KUKA KRL program: EPS_2_25694_RR02_A_20251117072404.src

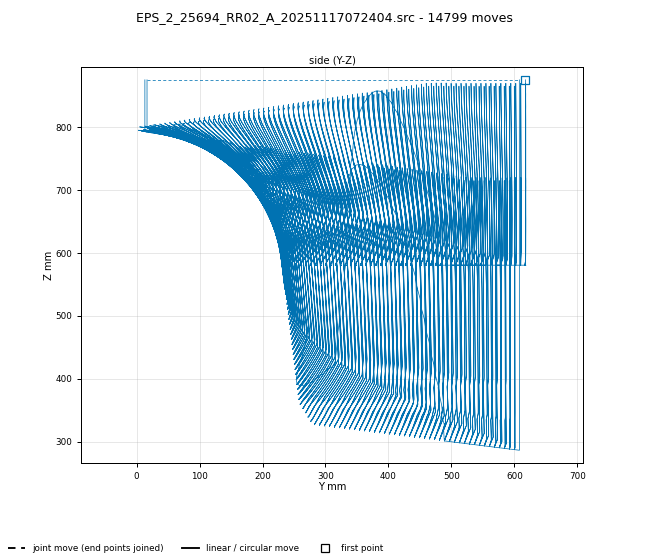
[picture p0: tool path of EPS_2_25694_RR02_A_20251117072404.src, 14799 of 14801 moves have a stored position in this frame; points joined in program order, loops and branches not executed]
&ACCESS RVP
&REL 4
&COMMENT QRS 19112012
&PARAM EDITMASK = *
DEF PART()
EXT BAS (BAS_COMMAND :IN,REAL :IN )
INT I
BAS (#INITMOV,0 )

;KUKA QRS Post kuka4.cps  Date:22-06-2017 !

File_ID=2908

QRS_PRE_INIT()

;Init var - Until changes are made in qrs_pre_init
Outlet_Square_prg=0
Inlet_1_Square_prg=0
Inlet_2_Square_prg=0
Inlet_3_Square_prg=0
Inlet_4_Square_prg=0
Inlet_5_Square_prg=0

Outlet_1={X 0.000, Y 466.000, Z 636.500, B 0.000, E1 0.000 }
Inlet_1={X 0.000, Y 521.440, Z 392.000, B 0.000, E1 180.000 }
Outlet_1_type=457
Inlet_1_type=366
;QRS#1=Sidecore dimensions
;QRS#2=450-18" Concrete
;QRS#3=375-15" PVC SDR 35
;QRS#4=
;QRS#5=
;QRS#6=
;QRS#7=
;QRS#8=
;QRS#9=28A PSX-2
;QRS#10=20Y PSX
;QRS#11=
;QRS#12=
;QRS#13=
;QRS#14=
;QRS#15=
;QRS#16=1220x127x1219 4'
;QRS#17=EPS Height
;QRS#18=865
;QRS#19=*
;QRS#20= UPDATED VERSION 22-06-2017
;QRS#21=*
Outlet_Square=0250
Inlet_1_Square=0250
Inlet_2_Square=0
Inlet_3_Square=0
Inlet_4_Square=0
Inlet_5_Square=0
Mill_Square=1
Outlet_Square_Prg=274
Inlet_1_Square_prg=252

QRS_INIT()

$ADVANCE=5

; T1
PTP {E1 171.23,E2 171.23}
PTP {X 0,Y 617.527,A -85,B 0,C 180,E1 171.23,E2 171.23,E3 0,E4 0,E5 0,E6 0}
QRS_SPEED_INIT()
LIN {X 0,Y 617.527,Z 875,A -85,B 0,C 180,E1 171.23,E2 171.23,E3 0,E4 0,E5 0,E6 0} C_VEL
LIN {X 0,Y 617.527,Z 582.66,A -85,B 0,C 180,E1 171.23,E2 171.23} C_VEL
LIN {X 0,Y 617.508,Z 580.66,A -85,B 0,C 180,E1 171.416,E2 171.416} C_VEL
LIN {X 0,Y 618.008,Z 580.66,A -85,B 0,C 180,E1 174.214,E2 174.214} C_VEL
LIN {X 0,Y 618.036,Z 580.66,A -85,B 0,C 180,E1 178.845,E2 178.845} C_VEL
LIN {X 0,Y 617.997,Z 580.66,A -85,B 0,C 180,E1 183.468,E2 183.468} C_VEL
LIN {X 0,Y 618.006,Z 580.66,A -85,B 0,C 180,E1 188.114,E2 188.114} C_VEL
LIN {X 0,Y 617.984,Z 580.66,A -85,B 0,C 180,E1 192.815,E2 192.815} C_VEL
LIN {X 0,Y 617.935,Z 580.66,A -85,B 0,C 180,E1 197.607,E2 197.607} C_VEL
LIN {X 0,Y 617.752,Z 580.66,A -85,B 0,C 180,E1 198.547,E2 198.547} C_VEL
LIN {X 0,Y 617.939,Z 580.66,A -85,B 0,C 180,E1 202.529,E2 202.529} C_VEL
LIN {X 0,Y 617.436,Z 580.66,A -85,B 0,C 180,E1 205.077,E2 205.077} C_VEL
LIN {X 0,Y 617.874,Z 580.66,A -85,B 0,C 180,E1 207.637,E2 207.637} C_VEL
LIN {X 0,Y 617.365,Z 580.66,A -85,B 0,C 180,E1 210.306,E2 210.306} C_VEL
LIN {X 0,Y 617.833,Z 580.66,A -85,B 0,C 180,E1 212.996,E2 212.996} C_VEL
LIN {X 0,Y 617.707,Z 580.66,A -85,B 0,C 180,E1 214.198,E2 214.198} C_VEL
LIN {X 0,Y 617.789,Z 580.66,A -85,B 0,C 180,E1 218.704,E2 218.704} C_VEL
LIN {X 0,Y 617.444,Z 580.66,A -85,B 0,C 180,E1 221.76,E2 221.76} C_VEL
LIN {X 0,Y 617.867,Z 580.66,A -85,B 0,C 180,E1 224.902,E2 224.902} C_VEL
LIN {X 0,Y 617.783,Z 580.66,A -85,B 0,C 180,E1 228.274,E2 228.274} C_VEL
LIN {X 0,Y 617.565,Z 580.66,A -85,B 0,C 180,E1 231.28,E2 231.28} C_VEL
LIN {X 0,Y 617.589,Z 580.66,A -85,B 0,C 180,E1 231.899,E2 231.899} C_VEL
LIN {X 0,Y 617.827,Z 580.66,A -85,B 0,C 180,E1 234.204,E2 234.204} C_VEL
LIN {X 0,Y 617.354,Z 580.66,A -85,B 0,C 180,E1 236.976,E2 236.976} C_VEL
LIN {X 0,Y 617.913,Z 580.66,A -85,B 0,C 180,E1 239.724,E2 239.724} C_VEL
LIN {X 0,Y 617.932,Z 580.66,A -85,B 0,C 180,E1 243.987,E2 243.987} C_VEL
LIN {X 0,Y 617.833,Z 580.66,A -85,B 0,C 180,E1 244.426,E2 244.426} C_VEL
LIN {X 0,Y 617.179,Z 580.66,A -85,B 0,C 180,E1 244.545,E2 244.545} C_VEL
LIN {X 0,Y 616.44,Z 580.66,A -85,B 0,C 180,E1 244.616,E2 244.616} C_VEL
LIN {X 0,Y 617.56,Z 586.788,A -85,B 0,C 180,E1 244.746,E2 244.746} C_VEL
LIN {X 0,Y 617.714,Z 589.526,A -85,B 0,C 180,E1 244.787,E2 244.787} C_VEL
LIN {X 0,Y 617.934,Z 647.055,A -85,B 0,C 180,E1 245.527,E2 245.527} C_VEL
LIN {X 0,Y 617.874,Z 657.74,A -85,B 0,C 180,E1 245.698,E2 245.698} C_VEL
LIN {X 0,Y 617.784,Z 666.504,A -85,B 0,C 180,E1 245.868,E2 245.868} C_VEL
LIN {X 0,Y 617.891,Z 680.089,A -85,B 0,C 180,E1 246.215,E2 246.215} C_VEL
LIN {X 0,Y 617.826,Z 690.542,A -85,B 0,C 180,E1 246.526,E2 246.526} C_VEL
LIN {X 0,Y 617.931,Z 702.898,A -85,B 0,C 180,E1 246.968,E2 246.968} C_VEL
LIN {X 0,Y 617.943,Z 713.369,A -85,B 0,C 180,E1 247.393,E2 247.393} C_VEL
LIN {X 0,Y 617.876,Z 723.673,A -85,B 0,C 180,E1 247.859,E2 247.859} C_VEL
LIN {X 0,Y 617.946,Z 734.342,A -85,B 0,C 180,E1 248.407,E2 248.407} C_VEL
LIN {X 0,Y 617.967,Z 745.217,A -85,B 0,C 180,E1 249.027,E2 249.027} C_VEL
LIN {X 0,Y 617.938,Z 755.025,A -85,B 0,C 180,E1 249.644,E2 249.644} C_VEL
LIN {X 0,Y 617.951,Z 764.531,A -85,B 0,C 180,E1 250.302,E2 250.302} C_VEL
LIN {X 0,Y 617.956,Z 773.726,A -85,B 0,C 180,E1 250.999,E2 250.999} C_VEL
LIN {X 0,Y 617.961,Z 782.652,A -85,B 0,C 180,E1 251.74,E2 251.74} C_VEL
LIN {X 0,Y 617.941,Z 791.031,A -85,B 0,C 180,E1 252.497,E2 252.497} C_VEL
LIN {X 0,Y 617.896,Z 798.423,A -85,B 0,C 180,E1 253.221,E2 253.221} C_VEL
LIN {X 0,Y 617.951,Z 806.122,A -85,B 0,C 180,E1 254.046,E2 254.046} C_VEL
LIN {X 0,Y 617.974,Z 812.663,A -85,B 0,C 180,E1 254.803,E2 254.803} C_VEL
LIN {X 0,Y 617.884,Z 819.775,A -85,B 0,C 180,E1 255.697,E2 255.697} C_VEL
LIN {X 0,Y 617.866,Z 826.241,A -85,B 0,C 180,E1 256.589,E2 256.589} C_VEL
LIN {X 0,Y 617.965,Z 832.101,A -85,B 0,C 180,E1 257.481,E2 257.481} C_VEL
LIN {X 0,Y 617.876,Z 837.462,A -85,B 0,C 180,E1 258.365,E2 258.365} C_VEL
LIN {X 0,Y 617.831,Z 843.765,A -85,B 0,C 180,E1 259.541,E2 259.541} C_VEL
LIN {X 0,Y 617.913,Z 847.328,A -85,B 0,C 180,E1 260.28,E2 260.28} C_VEL
LIN {X 0,Y 617.929,Z 852.365,A -85,B 0,C 180,E1 261.45,E2 261.45} C_VEL
LIN {X 0,Y 617.83,Z 855.756,A -85,B 0,C 180,E1 262.35,E2 262.35} C_VEL
LIN {X 0,Y 617.936,Z 860.149,A -85,B 0,C 180,E1 263.748,E2 263.748} C_VEL
LIN {X 0,Y 617.913,Z 862.617,A -85,B 0,C 180,E1 264.677,E2 264.677} C_VEL
LIN {X 0,Y 617.79,Z 864.668,A -85,B 0,C 180,E1 265.604,E2 265.604} C_VEL
LIN {X 0,Y 617.81,Z 866.258,A -85,B 0,C 180,E1 266.531,E2 266.531} C_VEL
LIN {X 0,Y 617.946,Z 867.44,A -85,B 0,C 180,E1 267.457,E2 267.457} C_VEL
LIN {X 0,Y 617.798,Z 868.661,A -85,B 0,C 180,E1 268.844,E2 268.844} C_VEL
LIN {X 0,Y 617.834,Z 868.908,A -85,B 0,C 180,E1 270.231,E2 270.231} C_VEL
LIN {X 0,Y 617.983,Z 868.61,A -85,B 0,C 180,E1 271.155,E2 271.155} C_VEL
LIN {X 0,Y 617.848,Z 867.993,A -85,B 0,C 180,E1 272.08,E2 272.08} C_VEL
LIN {X 0,Y 617.842,Z 866.25,A -85,B 0,C 180,E1 273.469,E2 273.469} C_VEL
LIN {X 0,Y 617.982,Z 864.618,A -85,B 0,C 180,E1 274.394,E2 274.394} C_VEL
LIN {X 0,Y 617.84,Z 862.637,A -85,B 0,C 180,E1 275.323,E2 275.323} C_VEL
LIN {X 0,Y 617.779,Z 860.19,A -85,B 0,C 180,E1 276.253,E2 276.253} C_VEL
LIN {X 0,Y 617.946,Z 855.729,A -85,B 0,C 180,E1 277.648,E2 277.648} C_VEL
LIN {X 0,Y 617.875,Z 851.344,A -85,B 0,C 180,E1 278.796,E2 278.796} C_VEL
LIN {X 0,Y 617.822,Z 847.617,A -85,B 0,C 180,E1 279.666,E2 279.666} C_VEL
LIN {X 0,Y 617.935,Z 842.259,A -85,B 0,C 180,E1 280.75,E2 280.75} C_VEL
LIN {X 0,Y 617.942,Z 837.451,A -85,B 0,C 180,E1 281.633,E2 281.633} C_VEL
LIN {X 0,Y 617.865,Z 830.2,A -85,B 0,C 180,E1 282.817,E2 282.817} C_VEL
LIN {X 0,Y 617.941,Z 824.139,A -85,B 0,C 180,E1 283.706,E2 283.706} C_VEL
LIN {X 0,Y 617.959,Z 817.472,A -85,B 0,C 180,E1 284.599,E2 284.599} C_VEL
LIN {X 0,Y 617.884,Z 809.504,A -85,B 0,C 180,E1 285.571,E2 285.571} C_VEL
LIN {X 0,Y 617.919,Z 802.445,A -85,B 0,C 180,E1 286.357,E2 286.357} C_VEL
LIN {X 0,Y 617.971,Z 794.292,A -85,B 0,C 180,E1 287.188,E2 287.188} C_VEL
LIN {X 0,Y 617.933,Z 787.152,A -85,B 0,C 180,E1 287.863,E2 287.863} C_VEL
LIN {X 0,Y 617.924,Z 778.254,A -85,B 0,C 180,E1 288.634,E2 288.634} C_VEL
LIN {X 0,Y 617.944,Z 769.358,A -85,B 0,C 180,E1 289.339,E2 289.339} C_VEL
LIN {X 0,Y 617.96,Z 760.867,A -85,B 0,C 180,E1 289.959,E2 289.959} C_VEL
LIN {X 0,Y 617.948,Z 751.476,A -85,B 0,C 180,E1 290.587,E2 290.587} C_VEL
LIN {X 0,Y 617.918,Z 741.285,A -85,B 0,C 180,E1 291.206,E2 291.206} C_VEL
LIN {X 0,Y 617.943,Z 731.422,A -85,B 0,C 180,E1 291.749,E2 291.749} C_VEL
LIN {X 0,Y 617.958,Z 720.367,A -85,B 0,C 180,E1 292.293,E2 292.293} C_VEL
LIN {X 0,Y 617.922,Z 709.607,A -85,B 0,C 180,E1 292.767,E2 292.767} C_VEL
LIN {X 0,Y 617.801,Z 699.701,A -85,B 0,C 180,E1 293.16,E2 293.16} C_VEL
LIN {X 0,Y 617.928,Z 686.719,A -85,B 0,C 180,E1 293.589,E2 293.589} C_VEL
LIN {X 0,Y 617.909,Z 674.953,A -85,B 0,C 180,E1 293.921,E2 293.921} C_VEL
LIN {X 0,Y 617.766,Z 663.559,A -85,B 0,C 180,E1 294.193,E2 294.193} C_VEL
LIN {X 0,Y 617.92,Z 651.868,A -85,B 0,C 180,E1 294.402,E2 294.402} C_VEL
LIN {X 0,Y 617.892,Z 634.191,A -85,B 0,C 180,E1 294.645,E2 294.645} C_VEL
LIN {X 0,Y 617.601,Z 587.358,A -85,B 0,C 180,E1 295.246,E2 295.246} C_VEL
LIN {X 0,Y 616.593,Z 581.43,A -85,B 0,C 180,E1 295.365,E2 295.365} C_VEL
LIN {X 0,Y 616.475,Z 580.66,A -85,B 0,C 180,E1 295.385,E2 295.385} C_VEL
LIN {X 0,Y 617.979,Z 580.66,A -85,B 0,C 180,E1 295.627,E2 295.627} C_VEL
LIN {X 0,Y 617.998,Z 580.66,A -85,B 0,C 180,E1 297.63,E2 297.63} C_VEL
LIN {X 0,Y 617.388,Z 580.66,A -85,B 0,C 180,E1 300.304,E2 300.304} C_VEL
LIN {X 0,Y 617.846,Z 580.66,A -85,B 0,C 180,E1 302.994,E2 302.994} C_VEL
LIN {X 0,Y 617.706,Z 580.66,A -85,B 0,C 180,E1 304.196,E2 304.196} C_VEL
LIN {X 0,Y 617.791,Z 580.66,A -85,B 0,C 180,E1 308.702,E2 308.702} C_VEL
LIN {X 0,Y 617.444,Z 580.66,A -85,B 0,C 180,E1 311.758,E2 311.758} C_VEL
LIN {X 0,Y 617.868,Z 580.66,A -85,B 0,C 180,E1 314.9,E2 314.9} C_VEL
LIN {X 0,Y 617.801,Z 580.66,A -85,B 0,C 180,E1 318.269,E2 318.269} C_VEL
LIN {X 0,Y 617.562,Z 580.66,A -85,B 0,C 180,E1 321.279,E2 321.279} C_VEL
LIN {X 0,Y 617.588,Z 580.66,A -85,B 0,C 180,E1 321.896,E2 321.896} C_VEL
LIN {X 0,Y 617.813,Z 580.66,A -85,B 0,C 180,E1 324.202,E2 324.202} C_VEL
LIN {X 0,Y 617.354,Z 580.66,A -85,B 0,C 180,E1 326.975,E2 326.975} C_VEL
LIN {X 0,Y 617.895,Z 580.66,A -85,B 0,C 180,E1 329.723,E2 329.723} C_VEL
LIN {X 0,Y 617.412,Z 580.66,A -85,B 0,C 180,E1 332.341,E2 332.341} C_VEL
LIN {X 0,Y 617.889,Z 580.66,A -85,B 0,C 180,E1 334.943,E2 334.943} C_VEL
LIN {X 0,Y 617.435,Z 580.66,A -85,B 0,C 180,E1 337.451,E2 337.451} C_VEL
LIN {X 0,Y 617.94,Z 580.66,A -85,B 0,C 180,E1 339.951,E2 339.951} C_VEL
LIN {X 0,Y 618.042,Z 580.66,A -85,B 0,C 180,E1 343.627,E2 343.627} C_VEL
LIN {X 0,Y 617.994,Z 580.66,A -85,B 0,C 180,E1 349.544,E2 349.544} C_VEL
LIN {X 0,Y 617.978,Z 580.66,A -85,B 0,C 180,E1 354.213,E2 354.213} C_VEL
LIN {X 0,Y 618.008,Z 580.66,A -85,B 0,C 180,E1 358.845,E2 358.845} C_VEL
LIN {X 0,Y 618.048,Z 580.66,A -85,B 0,C 180,E1 363.468,E2 363.468} C_VEL
LIN {X 0,Y 617.988,Z 580.66,A -85,B 0,C 180,E1 368.114,E2 368.114} C_VEL
LIN {X 0,Y 617.946,Z 580.66,A -85,B 0,C 180,E1 372.816,E2 372.816} C_VEL
LIN {X 0,Y 617.967,Z 580.66,A -85,B 0,C 180,E1 377.606,E2 377.606} C_VEL
LIN {X 0,Y 617.768,Z 580.66,A -85,B 0,C 180,E1 378.552,E2 378.552} C_VEL
LIN {X 0,Y 617.894,Z 580.66,A -85,B 0,C 180,E1 382.531,E2 382.531} C_VEL
LIN {X 0,Y 617.414,Z 580.66,A -85,B 0,C 180,E1 385.078,E2 385.078} C_VEL
LIN {X 0,Y 617.881,Z 580.66,A -85,B 0,C 180,E1 387.637,E2 387.637} C_VEL
LIN {X 0,Y 617.423,Z 580.66,A -85,B 0,C 180,E1 390.303,E2 390.303} C_VEL
LIN {X 0,Y 617.948,Z 580.66,A -85,B 0,C 180,E1 392.989,E2 392.989} C_VEL
LIN {X 0,Y 617.682,Z 580.66,A -85,B 0,C 180,E1 395.807,E2 395.807} C_VEL
LIN {X 0,Y 617.691,Z 580.66,A -85,B 0,C 180,E1 398.116,E2 398.116} C_VEL
LIN {X 0,Y 617.801,Z 580.66,A -85,B 0,C 180,E1 401.731,E2 401.731} C_VEL
LIN {X 0,Y 617.417,Z 580.66,A -85,B 0,C 180,E1 405.059,E2 405.059} C_VEL
LIN {X 0,Y 617.803,Z 580.66,A -85,B 0,C 180,E1 408.271,E2 408.271} C_VEL
LIN {X 0,Y 617.697,Z 580.66,A -85,B 0,C 180,E1 411.886,E2 411.886} C_VEL
LIN {X 0,Y 617.736,Z 580.66,A -85,B 0,C 180,E1 414.198,E2 414.198} C_VEL
LIN {X 0,Y 617.843,Z 580.66,A -85,B 0,C 180,E1 415.785,E2 415.785} C_VEL
LIN {X 0,Y 617.877,Z 580.66,A -85,B 0,C 180,E1 417.008,E2 417.008} C_VEL
LIN {X 0,Y 617.647,Z 580.66,A -85,B 0,C 180,E1 420.175,E2 420.175} C_VEL
LIN {X 0,Y 617.665,Z 580.66,A -85,B 0,C 180,E1 422.354,E2 422.354} C_VEL
LIN {X 0,Y 617.522,Z 580.66,A -85,B 0,C 180,E1 425.242,E2 425.242} C_VEL
LIN {X 0,Y 617.828,Z 580.66,A -85,B 0,C 180,E1 427.467,E2 427.467} C_VEL
LIN {X 0,Y 618.012,Z 580.66,A -85,B 0,C 180,E1 430.997,E2 430.997} C_VEL
LIN {X 0,Y 617.801,Z 580.749,A -85,B 0,C 180,E1 431.084,E2 431.084} C_VEL
LIN {X 0,Y 617.923,Z 591.91,A -85,B 0,C 180,E1 431.53,E2 431.53} C_VEL
LIN {X 0,Y 617.91,Z 600.741,A -85,B 0,C 180,E1 431.928,E2 431.928} C_VEL
LIN {X 0,Y 617.976,Z 609.876,A -85,B 0,C 180,E1 432.395,E2 432.395} C_VEL
LIN {X 0,Y 617.992,Z 617.77,A -85,B 0,C 180,E1 432.84,E2 432.84} C_VEL
LIN {X 0,Y 617.993,Z 624.968,A -85,B 0,C 180,E1 433.284,E2 433.284} C_VEL
LIN {X 0,Y 617.971,Z 633.892,A -85,B 0,C 180,E1 433.895,E2 433.895} C_VEL
LIN {X 0,Y 617.958,Z 641.958,A -85,B 0,C 180,E1 434.505,E2 434.505} C_VEL
LIN {X 0,Y 617.969,Z 649.146,A -85,B 0,C 180,E1 435.102,E2 435.102} C_VEL
LIN {X 0,Y 617.991,Z 655.741,A -85,B 0,C 180,E1 435.7,E2 435.7} C_VEL
LIN {X 0,Y 617.962,Z 663.24,A -85,B 0,C 180,E1 436.443,E2 436.443} C_VEL
LIN {X 0,Y 617.945,Z 670.024,A -85,B 0,C 180,E1 437.184,E2 437.184} C_VEL
LIN {X 0,Y 617.993,Z 677.361,A -85,B 0,C 180,E1 438.072,E2 438.072} C_VEL
LIN {X 0,Y 617.92,Z 683.858,A -85,B 0,C 180,E1 438.955,E2 438.955} C_VEL
LIN {X 0,Y 617.867,Z 688.987,A -85,B 0,C 180,E1 439.728,E2 439.728} C_VEL
LIN {X 0,Y 617.937,Z 694.438,A -85,B 0,C 180,E1 440.656,E2 440.656} C_VEL
LIN {X 0,Y 617.963,Z 698.446,A -85,B 0,C 180,E1 441.413,E2 441.413} C_VEL
LIN {X 0,Y 617.874,Z 702.863,A -85,B 0,C 180,E1 442.351,E2 442.351} C_VEL
LIN {X 0,Y 617.875,Z 704.864,A -85,B 0,C 180,E1 442.817,E2 442.817} C_VEL
LIN {X 0,Y 617.966,Z 708.364,A -85,B 0,C 180,E1 443.749,E2 443.749} C_VEL
LIN {X 0,Y 617.939,Z 711.343,A -85,B 0,C 180,E1 444.678,E2 444.678} C_VEL
LIN {X 0,Y 617.838,Z 713.822,A -85,B 0,C 180,E1 445.605,E2 445.605} C_VEL
LIN {X 0,Y 617.893,Z 715.764,A -85,B 0,C 180,E1 446.532,E2 446.532} C_VEL
LIN {X 0,Y 617.99,Z 717.213,A -85,B 0,C 180,E1 447.458,E2 447.458} C_VEL
LIN {X 0,Y 617.926,Z 717.776,A -85,B 0,C 180,E1 447.92,E2 447.92} C_VEL
LIN {X 0,Y 617.842,Z 718.587,A -85,B 0,C 180,E1 448.845,E2 448.845} C_VEL
LIN {X 0,Y 617.881,Z 718.907,A -85,B 0,C 180,E1 449.769,E2 449.769} C_VEL
LIN {X 0,Y 617.947,Z 718.867,A -85,B 0,C 180,E1 450.231,E2 450.231} C_VEL
LIN {X 0,Y 617.915,Z 718.503,A -85,B 0,C 180,E1 451.156,E2 451.156} C_VEL
LIN {X 0,Y 617.846,Z 717.146,A -85,B 0,C 180,E1 452.543,E2 452.543} C_VEL
LIN {X 0,Y 617.964,Z 715.592,A -85,B 0,C 180,E1 453.468,E2 453.468} C_VEL
LIN {X 0,Y 617.912,Z 713.595,A -85,B 0,C 180,E1 454.395,E2 454.395} C_VEL
LIN {X 0,Y 617.842,Z 711.097,A -85,B 0,C 180,E1 455.323,E2 455.323} C_VEL
LIN {X 0,Y 617.887,Z 708.049,A -85,B 0,C 180,E1 456.252,E2 456.252} C_VEL
LIN {X 0,Y 617.976,Z 704.45,A -85,B 0,C 180,E1 457.182,E2 457.182} C_VEL
LIN {X 0,Y 617.895,Z 700.32,A -85,B 0,C 180,E1 458.116,E2 458.116} C_VEL
LIN {X 0,Y 617.903,Z 695.375,A -85,B 0,C 180,E1 459.084,E2 459.084} C_VEL
LIN {X 0,Y 617.977,Z 690.86,A -85,B 0,C 180,E1 459.867,E2 459.867} C_VEL
LIN {X 0,Y 617.955,Z 687.19,A -85,B 0,C 180,E1 460.456,E2 460.456} C_VEL
LIN {X 0,Y 617.913,Z 682.18,A -85,B 0,C 180,E1 461.192,E2 461.192} C_VEL
LIN {X 0,Y 617.944,Z 676.638,A -85,B 0,C 180,E1 461.929,E2 461.929} C_VEL
LIN {X 0,Y 617.985,Z 670.528,A -85,B 0,C 180,E1 462.667,E2 462.667} C_VEL
LIN {X 0,Y 617.956,Z 663.803,A -85,B 0,C 180,E1 463.409,E2 463.409} C_VEL
LIN {X 0,Y 617.949,Z 657.931,A -85,B 0,C 180,E1 464.004,E2 464.004} C_VEL
LIN {X 0,Y 617.968,Z 651.535,A -85,B 0,C 180,E1 464.599,E2 464.599} C_VEL
LIN {X 0,Y 617.999,Z 644.545,A -85,B 0,C 180,E1 465.196,E2 465.196} C_VEL
LIN {X 0,Y 617.987,Z 637.134,A -85,B 0,C 180,E1 465.777,E2 465.777} C_VEL
LIN {X 0,Y 617.99,Z 628.688,A -85,B 0,C 180,E1 466.378,E2 466.378} C_VEL
LIN {X 0,Y 617.975,Z 620.778,A -85,B 0,C 180,E1 466.888,E2 466.888} C_VEL
LIN {X 0,Y 617.986,Z 613.859,A -85,B 0,C 180,E1 467.298,E2 467.298} C_VEL
LIN {X 0,Y 617.971,Z 605.435,A -85,B 0,C 180,E1 467.75,E2 467.75} C_VEL
LIN {X 0,Y 617.907,Z 596.414,A -85,B 0,C 180,E1 468.184,E2 468.184} C_VEL
LIN {X 0,Y 617.715,Z 586.549,A -85,B 0,C 180,E1 468.606,E2 468.606} C_VEL
LIN {X 0,Y 617.482,Z 580.66,A -85,B 0,C 180,E1 468.848,E2 468.848} C_VEL
LIN {X 0,Y 617.844,Z 580.66,A -85,B 0,C 180,E1 468.93,E2 468.93} C_VEL
LIN {X 0,Y 618.044,Z 580.66,A -85,B 0,C 180,E1 469.031,E2 469.031} C_VEL
LIN {X 0,Y 618.046,Z 580.66,A -85,B 0,C 180,E1 470.045,E2 470.045} C_VEL
LIN {X 0,Y 617.926,Z 580.66,A -85,B 0,C 180,E1 475.055,E2 475.055} C_VEL
LIN {X 0,Y 617.412,Z 580.66,A -85,B 0,C 180,E1 477.659,E2 477.659} C_VEL
LIN {X 0,Y 617.854,Z 580.66,A -85,B 0,C 180,E1 480.279,E2 480.279} C_VEL
LIN {X 0,Y 617.333,Z 580.66,A -85,B 0,C 180,E1 483.025,E2 483.025} C_VEL
LIN {X 0,Y 617.818,Z 580.66,A -85,B 0,C 180,E1 485.797,E2 485.797} C_VEL
LIN {X 0,Y 617.907,Z 580.66,A -85,B 0,C 180,E1 488.694,E2 488.694} C_VEL
LIN {X 0,Y 617.42,Z 580.66,A -85,B 0,C 180,E1 491.761,E2 491.761} C_VEL
LIN {X 0,Y 617.838,Z 580.66,A -85,B 0,C 180,E1 494.903,E2 494.903} C_VEL
LIN {X 0,Y 617.754,Z 580.66,A -85,B 0,C 180,E1 498.275,E2 498.275} C_VEL
LIN {X 0,Y 617.542,Z 580.66,A -85,B 0,C 180,E1 501.278,E2 501.278} C_VEL
LIN {X 0,Y 617.816,Z 580.66,A -85,B 0,C 180,E1 504.202,E2 504.202} C_VEL
LIN {X 0,Y 617.317,Z 580.66,A -85,B 0,C 180,E1 506.973,E2 506.973} C_VEL
LIN {X 0,Y 617.842,Z 580.66,A -85,B 0,C 180,E1 509.72,E2 509.72} C_VEL
LIN {X 0,Y 617.389,Z 580.66,A -85,B 0,C 180,E1 512.339,E2 512.339} C_VEL
LIN {X 0,Y 617.892,Z 580.66,A -85,B 0,C 180,E1 514.943,E2 514.943} C_VEL
LIN {X 0,Y 617.441,Z 580.66,A -85,B 0,C 180,E1 517.452,E2 517.452} C_VEL
LIN {X 0,Y 617.945,Z 580.66,A -85,B 0,C 180,E1 519.951,E2 519.951} C_VEL
LIN {X 0,Y 618.009,Z 580.66,A -85,B 0,C 180,E1 523.636,E2 523.636} C_VEL
LIN {X 0,Y 617.95,Z 580.66,A -85,B 0,C 180,E1 529.543,E2 529.543} C_VEL
LIN {X 0,Y 617.508,Z 580.66,A -85,B 0,C 180,E1 531.416,E2 531.416} C_VEL
LIN {X 0,Y 613.842,Z 580.66,A -85,B 0,C 180,E1 533.008,E2 533.008} C_VEL
LIN {X 0,Y 609.952,Z 580.66,A -85,B 0,C 180,E1 534.619,E2 534.619} C_VEL
LIN {X 0,Y 609.775,Z 580.66,A -85,B 0,C 180,E1 539.996,E2 539.996} C_VEL
LIN {X 0,Y 609.835,Z 580.66,A -85,B 0,C 180,E1 544.267,E2 544.267} C_VEL
LIN {X 0,Y 609.932,Z 580.66,A -85,B 0,C 180,E1 548.561,E2 548.561} C_VEL
LIN {X 0,Y 610.054,Z 580.66,A -85,B 0,C 180,E1 552.902,E2 552.902} C_VEL
LIN {X 0,Y 609.793,Z 580.66,A -85,B 0,C 180,E1 558.826,E2 558.826} C_VEL
LIN {X 0,Y 609.731,Z 580.66,A -85,B 0,C 180,E1 563.405,E2 563.405} C_VEL
LIN {X 0,Y 609.791,Z 580.66,A -85,B 0,C 180,E1 568.143,E2 568.143} C_VEL
LIN {X 0,Y 609.938,Z 580.66,A -85,B 0,C 180,E1 573.095,E2 573.095} C_VEL
LIN {X 0,Y 609.609,Z 580.66,A -85,B 0,C 180,E1 579.652,E2 579.652} C_VEL
LIN {X 0,Y 609.721,Z 580.66,A -85,B 0,C 180,E1 585.949,E2 585.949} C_VEL
LIN {X 0,Y 609.565,Z 580.66,A -85,B 0,C 180,E1 590.345,E2 590.345} C_VEL
LIN {X 0,Y 609.614,Z 580.66,A -85,B 0,C 180,E1 595.163,E2 595.163} C_VEL
LIN {X 0,Y 609.814,Z 580.66,A -85,B 0,C 180,E1 600.331,E2 600.331} C_VEL
LIN {X 0,Y 609.422,Z 580.66,A -85,B 0,C 180,E1 604.278,E2 604.278} C_VEL
LIN {X 0,Y 610.603,Z 601.613,A -85,B 0,C 180,E1 604.626,E2 604.626} C_VEL
LIN {X 0,Y 610.594,Z 666.131,A -85,B 0,C 180,E1 605.557,E2 605.557} C_VEL
LIN {X 0,Y 610.606,Z 702.84,A -85,B 0,C 180,E1 606.673,E2 606.673} C_VEL
LIN {X 0,Y 610.469,Z 736.562,A -85,B 0,C 180,E1 608.254,E2 608.254} C_VEL
LIN {X 0,Y 610.341,Z 768.501,A -85,B 0,C 180,E1 610.345,E2 610.345} C_VEL
LIN {X 0,Y 610.22,Z 797.222,A -85,B 0,C 180,E1 612.863,E2 612.863} C_VEL
LIN {X 0,Y 610.116,Z 822.296,A -85,B 0,C 180,E1 615.814,E2 615.814} C_VEL
LIN {X 0,Y 610.041,Z 841.765,A -85,B 0,C 180,E1 618.909,E2 618.909} C_VEL
LIN {X 0,Y 610.029,Z 856.171,A -85,B 0,C 180,E1 622.153,E2 622.153} C_VEL
LIN {X 0,Y 610.029,Z 864.449,A -85,B 0,C 180,E1 625.015,E2 625.015} C_VEL
LIN {X 0,Y 609.996,Z 869.506,A -85,B 0,C 180,E1 628.576,E2 628.576} C_VEL
LIN {X 0,Y 610.121,Z 869.508,A -85,B 0,C 180,E1 631.421,E2 631.421} C_VEL
LIN {X 0,Y 610.052,Z 864.454,A -85,B 0,C 180,E1 634.982,E2 634.982} C_VEL
LIN {X 0,Y 610.08,Z 853.503,A -85,B 0,C 180,E1 638.562,E2 638.562} C_VEL
LIN {X 0,Y 610.103,Z 836.72,A -85,B 0,C 180,E1 641.994,E2 641.994} C_VEL
LIN {X 0,Y 610.174,Z 815.251,A -85,B 0,C 180,E1 645.103,E2 645.103} C_VEL
LIN {X 0,Y 610.254,Z 788.597,A -85,B 0,C 180,E1 647.972,E2 647.972} C_VEL
LIN {X 0,Y 610.393,Z 758.021,A -85,B 0,C 180,E1 650.413,E2 650.413} C_VEL
LIN {X 0,Y 610.532,Z 725.757,A -85,B 0,C 180,E1 652.315,E2 652.315} C_VEL
LIN {X 0,Y 610.645,Z 690.377,A -85,B 0,C 180,E1 653.772,E2 653.772} C_VEL
LIN {X 0,Y 610.725,Z 653.833,A -85,B 0,C 180,E1 654.679,E2 654.679} C_VEL
LIN {X 0,Y 609.77,Z 584.389,A -85,B 0,C 180,E1 655.631,E2 655.631} C_VEL
LIN {X 0,Y 609.682,Z 580.66,A -85,B 0,C 180,E1 655.757,E2 655.757} C_VEL
LIN {X 0,Y 609.507,Z 580.66,A -85,B 0,C 180,E1 659.787,E2 659.787} C_VEL
LIN {X 0,Y 609.945,Z 580.66,A -85,B 0,C 180,E1 663.097,E2 663.097} C_VEL
LIN {X 0,Y 609.593,Z 580.66,A -85,B 0,C 180,E1 669.658,E2 669.658} C_VEL
LIN {X 0,Y 609.734,Z 580.66,A -85,B 0,C 180,E1 675.957,E2 675.957} C_VEL
LIN {X 0,Y 609.567,Z 580.66,A -85,B 0,C 180,E1 680.349,E2 680.349} C_VEL
LIN {X 0,Y 609.607,Z 580.66,A -85,B 0,C 180,E1 685.169,E2 685.169} C_VEL
LIN {X 0,Y 609.783,Z 580.66,A -85,B 0,C 180,E1 690.341,E2 690.341} C_VEL
LIN {X 0,Y 609.961,Z 580.66,A -85,B 0,C 180,E1 695.045,E2 695.045} C_VEL
LIN {X 0,Y 609.793,Z 580.66,A -85,B 0,C 180,E1 701.174,E2 701.174} C_VEL
LIN {X 0,Y 609.393,Z 580.66,A -85,B 0,C 180,E1 705.678,E2 705.678} C_VEL
LIN {X 0,Y 609.919,Z 580.66,A -85,B 0,C 180,E1 709.997,E2 709.997} C_VEL
LIN {X 0,Y 610.056,Z 580.66,A -85,B 0,C 180,E1 714.307,E2 714.307} C_VEL
LIN {X 0,Y 609.744,Z 580.66,A -85,B 0,C 180,E1 720.004,E2 720.004} C_VEL
LIN {X 0,Y 609.85,Z 580.66,A -85,B 0,C 180,E1 724.275,E2 724.275} C_VEL
LIN {X 0,Y 609.914,Z 580.66,A -85,B 0,C 180,E1 728.57,E2 728.57} C_VEL
LIN {X 0,Y 609.999,Z 580.66,A -85,B 0,C 180,E1 732.912,E2 732.912} C_VEL
LIN {X 0,Y 609.783,Z 580.66,A -85,B 0,C 180,E1 738.835,E2 738.835} C_VEL
LIN {X 0,Y 609.7,Z 580.66,A -85,B 0,C 180,E1 743.415,E2 743.415} C_VEL
LIN {X 0,Y 609.795,Z 580.66,A -85,B 0,C 180,E1 748.152,E2 748.152} C_VEL
LIN {X 0,Y 610.006,Z 580.66,A -85,B 0,C 180,E1 753.1,E2 753.1} C_VEL
LIN {X 0,Y 609.73,Z 580.66,A -85,B 0,C 180,E1 758.378,E2 758.378} C_VEL
LIN {X 0,Y 609.77,Z 580.66,A -85,B 0,C 180,E1 762.103,E2 762.103} C_VEL
LIN {X 0,Y 609.865,Z 580.66,A -85,B 0,C 180,E1 768.145,E2 768.145} C_VEL
LIN {X 0,Y 609.733,Z 580.66,A -85,B 0,C 180,E1 773.422,E2 773.422} C_VEL
LIN {X 0,Y 609.795,Z 580.66,A -85,B 0,C 180,E1 777.59,E2 777.59} C_VEL
LIN {X 0,Y 609.7,Z 580.66,A -85,B 0,C 180,E1 781.85,E2 781.85} C_VEL
LIN {X 0,Y 609.813,Z 580.66,A -85,B 0,C 180,E1 788.137,E2 788.137} C_VEL
LIN {X 0,Y 610.063,Z 580.755,A -85,B 0,C 180,E1 790.836,E2 790.836} C_VEL
LIN {X 0,Y 610.376,Z 612.485,A -85,B 0,C 180,E1 792.312,E2 792.312} C_VEL
LIN {X 0,Y 610.257,Z 642.503,A -85,B 0,C 180,E1 794.338,E2 794.338} C_VEL
LIN {X 0,Y 610.2,Z 667.86,A -85,B 0,C 180,E1 796.733,E2 796.733} C_VEL
LIN {X 0,Y 610.105,Z 688.675,A -85,B 0,C 180,E1 799.456,E2 799.456} C_VEL
LIN {X 0,Y 610.08,Z 704.253,A -85,B 0,C 180,E1 802.397,E2 802.397} C_VEL
LIN {X 0,Y 610.06,Z 713.378,A -85,B 0,C 180,E1 805.018,E2 805.018} C_VEL
LIN {X 0,Y 610.125,Z 717.884,A -85,B 0,C 180,E1 807.157,E2 807.157} C_VEL
LIN {X 0,Y 610.088,Z 719.996,A -85,B 0,C 180,E1 810.001,E2 810.001} C_VEL
LIN {X 0,Y 610.04,Z 717.729,A -85,B 0,C 180,E1 812.846,E2 812.846} C_VEL
LIN {X 0,Y 610.068,Z 709.867,A -85,B 0,C 180,E1 816.056,E2 816.056} C_VEL
LIN {X 0,Y 610.101,Z 697.553,A -85,B 0,C 180,E1 818.924,E2 818.924} C_VEL
LIN {X 0,Y 610.144,Z 679.155,A -85,B 0,C 180,E1 821.814,E2 821.814} C_VEL
LIN {X 0,Y 610.218,Z 655.502,A -85,B 0,C 180,E1 824.441,E2 824.441} C_VEL
LIN {X 0,Y 610.329,Z 627.575,A -85,B 0,C 180,E1 826.669,E2 826.669} C_VEL
LIN {X 0,Y 610.345,Z 595.936,A -85,B 0,C 180,E1 828.439,E2 828.439} C_VEL
LIN {X 0,Y 610.16,Z 580.66,A -85,B 0,C 180,E1 829.133,E2 829.133} C_VEL
LIN {X 0,Y 609.998,Z 580.66,A -85,B 0,C 180,E1 834.959,E2 834.959} C_VEL
LIN {X 0,Y 609.796,Z 580.66,A -85,B 0,C 180,E1 839.775,E2 839.775} C_VEL
LIN {X 0,Y 609.79,Z 580.66,A -85,B 0,C 180,E1 846.577,E2 846.577} C_VEL
LIN {X 0,Y 609.542,Z 580.66,A -85,B 0,C 180,E1 850.228,E2 850.228} C_VEL
LIN {X 0,Y 609.675,Z 580.66,A -85,B 0,C 180,E1 856.07,E2 856.07} C_VEL
LIN {X 0,Y 609.528,Z 580.66,A -85,B 0,C 180,E1 860.357,E2 860.357} C_VEL
LIN {X 0,Y 609.596,Z 580.66,A -85,B 0,C 180,E1 865.158,E2 865.158} C_VEL
LIN {X 0,Y 609.742,Z 580.66,A -85,B 0,C 180,E1 870.353,E2 870.353} C_VEL
LIN {X 0,Y 609.98,Z 580.66,A -85,B 0,C 180,E1 875.038,E2 875.038} C_VEL
LIN {X 0,Y 609.814,Z 580.66,A -85,B 0,C 180,E1 881.166,E2 881.166} C_VEL
LIN {X 0,Y 609.34,Z 580.66,A -85,B 0,C 180,E1 885.708,E2 885.708} C_VEL
LIN {X 0,Y 609.891,Z 580.66,A -85,B 0,C 180,E1 889.989,E2 889.989} C_VEL
LIN {X 0,Y 609.952,Z 580.66,A -85,B 0,C 180,E1 894.619,E2 894.619} C_VEL
LIN {X 0,Y 605.699,Z 580.66,A -85,B 0,C 180,E1 896.215,E2 896.215} C_VEL
LIN {X 0,Y 601.911,Z 580.66,A -85,B 0,C 180,E1 897.833,E2 897.833} C_VEL
LIN {X 0,Y 601.976,Z 580.66,A -85,B 0,C 180,E1 902.879,E2 902.879} C_VEL
LIN {X 0,Y 601.99,Z 580.66,A -85,B 0,C 180,E1 908.675,E2 908.675} C_VEL
LIN {X 0,Y 602.076,Z 580.66,A -85,B 0,C 180,E1 913.076,E2 913.076} C_VEL
LIN {X 0,Y 601.84,Z 580.66,A -85,B 0,C 180,E1 919.085,E2 919.085} C_VEL
LIN {X 0,Y 601.755,Z 580.66,A -85,B 0,C 180,E1 923.734,E2 923.734} C_VEL
LIN {X 0,Y 601.771,Z 580.66,A -85,B 0,C 180,E1 928.552,E2 928.552} C_VEL
LIN {X 0,Y 601.82,Z 580.66,A -85,B 0,C 180,E1 933.879,E2 933.879} C_VEL
LIN {X 0,Y 601.76,Z 580.66,A -85,B 0,C 180,E1 938.971,E2 938.971} C_VEL
LIN {X 0,Y 601.731,Z 580.66,A -85,B 0,C 180,E1 945.208,E2 945.208} C_VEL
LIN {X 0,Y 601.737,Z 580.66,A -85,B 0,C 180,E1 951.253,E2 951.253} C_VEL
LIN {X 0,Y 601.54,Z 580.66,A -85,B 0,C 180,E1 956.376,E2 956.376} C_VEL
LIN {X 0,Y 601.737,Z 580.66,A -85,B 0,C 180,E1 961.71,E2 961.71} C_VEL
LIN {X 0,Y 601.847,Z 580.66,A -85,B 0,C 180,E1 963.958,E2 963.958} C_VEL
LIN {X 0,Y 603.468,Z 597.745,A -85,B 0,C 180,E1 964.255,E2 964.255} C_VEL
LIN {X 0,Y 603.4,Z 666.109,A -85,B 0,C 180,E1 965.245,E2 965.245} C_VEL
LIN {X 0,Y 603.293,Z 702.843,A -85,B 0,C 180,E1 966.373,E2 966.373} C_VEL
LIN {X 0,Y 603.024,Z 737.402,A -85,B 0,C 180,E1 968.02,E2 968.02} C_VEL
LIN {X 0,Y 602.743,Z 769.05,A -85,B 0,C 180,E1 970.129,E2 970.129} C_VEL
LIN {X 0,Y 602.475,Z 799.299,A -85,B 0,C 180,E1 972.858,E2 972.858} C_VEL
LIN {X 0,Y 602.308,Z 823.634,A -85,B 0,C 180,E1 975.812,E2 975.812} C_VEL
LIN {X 0,Y 602.183,Z 842.817,A -85,B 0,C 180,E1 978.959,E2 978.959} C_VEL
LIN {X 0,Y 602.139,Z 857.455,A -85,B 0,C 180,E1 982.413,E2 982.413} C_VEL
LIN {X 0,Y 602.094,Z 865.968,A -85,B 0,C 180,E1 985.672,E2 985.672} C_VEL
LIN {X 0,Y 602.096,Z 869.506,A -85,B 0,C 180,E1 988.558,E2 988.558} C_VEL
LIN {X 0,Y 602.216,Z 869.508,A -85,B 0,C 180,E1 991.439,E2 991.439} C_VEL
LIN {X 0,Y 602.161,Z 864.455,A -85,B 0,C 180,E1 995.047,E2 995.047} C_VEL
LIN {X 0,Y 602.185,Z 853.503,A -85,B 0,C 180,E1 998.675,E2 998.675} C_VEL
LIN {X 0,Y 602.248,Z 836.721,A -85,B 0,C 180,E1 1002.153,E2 1002.153} C_VEL
LIN {X 0,Y 602.382,Z 815.277,A -85,B 0,C 180,E1 1005.301,E2 1005.301} C_VEL
LIN {X 0,Y 602.598,Z 788.598,A -85,B 0,C 180,E1 1008.208,E2 1008.208} C_VEL
LIN {X 0,Y 602.858,Z 757.351,A -85,B 0,C 180,E1 1010.727,E2 1010.727} C_VEL
LIN {X 0,Y 603.16,Z 723.319,A -85,B 0,C 180,E1 1012.729,E2 1012.729} C_VEL
LIN {X 0,Y 603.399,Z 687.811,A -85,B 0,C 180,E1 1014.16,E2 1014.16} C_VEL
LIN {X 0,Y 603.546,Z 653.817,A -85,B 0,C 180,E1 1014.993,E2 1014.993} C_VEL
LIN {X 0,Y 602.7,Z 585.728,A -85,B 0,C 180,E1 1015.936,E2 1015.936} C_VEL
LIN {X 0,Y 601.937,Z 580.66,A -85,B 0,C 180,E1 1016.114,E2 1016.114} C_VEL
LIN {X 0,Y 601.72,Z 580.66,A -85,B 0,C 180,E1 1021.895,E2 1021.895} C_VEL
LIN {X 0,Y 601.552,Z 580.66,A -85,B 0,C 180,E1 1027.158,E2 1027.158} C_VEL
LIN {X 0,Y 601.568,Z 580.66,A -85,B 0,C 180,E1 1030.977,E2 1030.977} C_VEL
LIN {X 0,Y 601.772,Z 580.66,A -85,B 0,C 180,E1 1036.853,E2 1036.853} C_VEL
LIN {X 0,Y 601.771,Z 580.66,A -85,B 0,C 180,E1 1042.86,E2 1042.86} C_VEL
LIN {X 0,Y 601.728,Z 580.66,A -85,B 0,C 180,E1 1048.81,E2 1048.81} C_VEL
LIN {X 0,Y 602.001,Z 580.66,A -85,B 0,C 180,E1 1054.873,E2 1054.873} C_VEL
LIN {X 0,Y 601.936,Z 580.66,A -85,B 0,C 180,E1 1060.918,E2 1060.918} C_VEL
LIN {X 0,Y 601.542,Z 580.66,A -85,B 0,C 180,E1 1065.427,E2 1065.427} C_VEL
LIN {X 0,Y 601.976,Z 580.66,A -85,B 0,C 180,E1 1069.864,E2 1069.864} C_VEL
LIN {X 0,Y 602.146,Z 580.66,A -85,B 0,C 180,E1 1074.232,E2 1074.232} C_VEL
LIN {X 0,Y 601.844,Z 580.66,A -85,B 0,C 180,E1 1080.004,E2 1080.004} C_VEL
LIN {X 0,Y 601.962,Z 580.66,A -85,B 0,C 180,E1 1084.331,E2 1084.331} C_VEL
LIN {X 0,Y 601.972,Z 580.66,A -85,B 0,C 180,E1 1088.684,E2 1088.684} C_VEL
LIN {X 0,Y 602.027,Z 580.66,A -85,B 0,C 180,E1 1093.086,E2 1093.086} C_VEL
LIN {X 0,Y 602.015,Z 580.66,A -85,B 0,C 180,E1 1097.569,E2 1097.569} C_VEL
LIN {X 0,Y 601.725,Z 580.66,A -85,B 0,C 180,E1 1103.744,E2 1103.744} C_VEL
LIN {X 0,Y 601.785,Z 580.66,A -85,B 0,C 180,E1 1108.561,E2 1108.561} C_VEL
LIN {X 0,Y 601.91,Z 580.66,A -85,B 0,C 180,E1 1113.897,E2 1113.897} C_VEL
LIN {X 0,Y 601.722,Z 580.66,A -85,B 0,C 180,E1 1118.984,E2 1118.984} C_VEL
LIN {X 0,Y 601.602,Z 580.66,A -85,B 0,C 180,E1 1123.13,E2 1123.13} C_VEL
LIN {X 0,Y 601.731,Z 580.66,A -85,B 0,C 180,E1 1129.144,E2 1129.144} C_VEL
LIN {X 0,Y 601.883,Z 580.66,A -85,B 0,C 180,E1 1134.652,E2 1134.652} C_VEL
LIN {X 0,Y 601.77,Z 580.66,A -85,B 0,C 180,E1 1139.79,E2 1139.79} C_VEL
LIN {X 0,Y 601.715,Z 580.66,A -85,B 0,C 180,E1 1144.944,E2 1144.944} C_VEL
LIN {X 0,Y 602.101,Z 581.093,A -85,B 0,C 180,E1 1150.587,E2 1150.587} C_VEL
LIN {X 0,Y 602.777,Z 612.479,A -85,B 0,C 180,E1 1152.081,E2 1152.081} C_VEL
LIN {X 0,Y 602.569,Z 642.629,A -85,B 0,C 180,E1 1154.144,E2 1154.144} C_VEL
LIN {X 0,Y 602.404,Z 667.855,A -85,B 0,C 180,E1 1156.558,E2 1156.558} C_VEL
LIN {X 0,Y 602.23,Z 688.273,A -85,B 0,C 180,E1 1159.256,E2 1159.256} C_VEL
LIN {X 0,Y 602.202,Z 703.222,A -85,B 0,C 180,E1 1162.053,E2 1162.053} C_VEL
LIN {X 0,Y 602.171,Z 713.377,A -85,B 0,C 180,E1 1164.953,E2 1164.953} C_VEL
LIN {X 0,Y 602.22,Z 717.884,A -85,B 0,C 180,E1 1167.119,E2 1167.119} C_VEL
LIN {X 0,Y 602.188,Z 719.996,A -85,B 0,C 180,E1 1170.001,E2 1170.001} C_VEL
LIN {X 0,Y 602.146,Z 717.731,A -85,B 0,C 180,E1 1172.884,E2 1172.884} C_VEL
LIN {X 0,Y 602.174,Z 711.013,A -85,B 0,C 180,E1 1175.773,E2 1175.773} C_VEL
LIN {X 0,Y 602.21,Z 699.392,A -85,B 0,C 180,E1 1178.677,E2 1178.677} C_VEL
LIN {X 0,Y 602.297,Z 681.829,A -85,B 0,C 180,E1 1181.603,E2 1181.603} C_VEL
LIN {X 0,Y 602.445,Z 660.096,A -85,B 0,C 180,E1 1184.185,E2 1184.185} C_VEL
LIN {X 0,Y 602.659,Z 632.798,A -85,B 0,C 180,E1 1186.524,E2 1186.524} C_VEL
LIN {X 0,Y 602.786,Z 601.859,A -85,B 0,C 180,E1 1188.394,E2 1188.394} C_VEL
LIN {X 0,Y 602.253,Z 580.66,A -85,B 0,C 180,E1 1189.348,E2 1189.348} C_VEL
LIN {X 0,Y 601.981,Z 580.66,A -85,B 0,C 180,E1 1195.314,E2 1195.314} C_VEL
LIN {X 0,Y 601.711,Z 580.66,A -85,B 0,C 180,E1 1201.176,E2 1201.176} C_VEL
LIN {X 0,Y 601.871,Z 580.66,A -85,B 0,C 180,E1 1207.139,E2 1207.139} C_VEL
LIN {X 0,Y 601.596,Z 580.66,A -85,B 0,C 180,E1 1213.121,E2 1213.121} C_VEL
LIN {X 0,Y 601.728,Z 580.66,A -85,B 0,C 180,E1 1219.013,E2 1219.013} C_VEL
LIN {X 0,Y 601.703,Z 580.66,A -85,B 0,C 180,E1 1224.633,E2 1224.633} C_VEL
LIN {X 0,Y 601.761,Z 580.66,A -85,B 0,C 180,E1 1229.784,E2 1229.784} C_VEL
LIN {X 0,Y 602.029,Z 580.66,A -85,B 0,C 180,E1 1234.873,E2 1234.873} C_VEL
LIN {X 0,Y 601.942,Z 580.66,A -85,B 0,C 180,E1 1240.91,E2 1240.91} C_VEL
LIN {X 0,Y 601.515,Z 580.66,A -85,B 0,C 180,E1 1245.418,E2 1245.418} C_VEL
LIN {X 0,Y 601.945,Z 580.66,A -85,B 0,C 180,E1 1249.855,E2 1249.855} C_VEL
LIN {X 0,Y 602.03,Z 580.66,A -85,B 0,C 180,E1 1254.596,E2 1254.596} C_VEL
LIN {X 0,Y 601.911,Z 580.66,A -85,B 0,C 180,E1 1257.833,E2 1257.833} C_VEL
LIN {X 0,Y 599.465,Z 580.66,A -85,B 0,C 180,E1 1259.063,E2 1259.063} C_VEL
LIN {X 0,Y 593.926,Z 580.66,A -85,B 0,C 180,E1 1260.901,E2 1260.901} C_VEL
LIN {X 0,Y 593.823,Z 580.66,A -85,B 0,C 180,E1 1261.114,E2 1261.114} C_VEL
LIN {X 0,Y 593.849,Z 580.66,A -85,B 0,C 180,E1 1266.105,E2 1266.105} C_VEL
LIN {X 0,Y 593.811,Z 580.66,A -85,B 0,C 180,E1 1270.277,E2 1270.277} C_VEL
LIN {X 0,Y 593.787,Z 580.66,A -85,B 0,C 180,E1 1274.768,E2 1274.768} C_VEL
LIN {X 0,Y 593.884,Z 580.66,A -85,B 0,C 180,E1 1279.39,E2 1279.39} C_VEL
LIN {X 0,Y 593.829,Z 580.66,A -85,B 0,C 180,E1 1284.071,E2 1284.071} C_VEL
LIN {X 0,Y 593.765,Z 580.66,A -85,B 0,C 180,E1 1288.974,E2 1288.974} C_VEL
LIN {X 0,Y 593.879,Z 580.66,A -85,B 0,C 180,E1 1294.111,E2 1294.111} C_VEL
LIN {X 0,Y 593.682,Z 580.66,A -85,B 0,C 180,E1 1300.085,E2 1300.085} C_VEL
LIN {X 0,Y 593.798,Z 580.66,A -85,B 0,C 180,E1 1305.549,E2 1305.549} C_VEL
LIN {X 0,Y 593.741,Z 580.66,A -85,B 0,C 180,E1 1310.393,E2 1310.393} C_VEL
LIN {X 0,Y 593.674,Z 580.66,A -85,B 0,C 180,E1 1315.87,E2 1315.87} C_VEL
LIN {X 0,Y 593.822,Z 580.66,A -85,B 0,C 180,E1 1321.023,E2 1321.023} C_VEL
LIN {X 0,Y 593.976,Z 580.66,A -85,B 0,C 180,E1 1323.579,E2 1323.579} C_VEL
LIN {X 0,Y 596.348,Z 595.229,A -85,B 0,C 180,E1 1323.891,E2 1323.891} C_VEL
LIN {X 0,Y 596.217,Z 665.817,A -85,B 0,C 180,E1 1324.92,E2 1324.92} C_VEL
LIN {X 0,Y 595.974,Z 702.661,A -85,B 0,C 180,E1 1326.058,E2 1326.058} C_VEL
LIN {X 0,Y 595.571,Z 736.631,A -85,B 0,C 180,E1 1327.685,E2 1327.685} C_VEL
LIN {X 0,Y 595.182,Z 768.999,A -85,B 0,C 180,E1 1329.861,E2 1329.861} C_VEL
LIN {X 0,Y 594.794,Z 798.342,A -85,B 0,C 180,E1 1332.526,E2 1332.526} C_VEL
LIN {X 0,Y 594.503,Z 822.969,A -85,B 0,C 180,E1 1335.528,E2 1335.528} C_VEL
LIN {X 0,Y 594.333,Z 842.002,A -85,B 0,C 180,E1 1338.657,E2 1338.657} C_VEL
LIN {X 0,Y 594.29,Z 856.172,A -85,B 0,C 180,E1 1341.944,E2 1341.944} C_VEL
LIN {X 0,Y 594.269,Z 864.45,A -85,B 0,C 180,E1 1344.883,E2 1344.883} C_VEL
LIN {X 0,Y 594.195,Z 869.507,A -85,B 0,C 180,E1 1348.539,E2 1348.539} C_VEL
LIN {X 0,Y 594.311,Z 869.508,A -85,B 0,C 180,E1 1351.458,E2 1351.458} C_VEL
LIN {X 0,Y 594.283,Z 864.455,A -85,B 0,C 180,E1 1355.114,E2 1355.114} C_VEL
LIN {X 0,Y 594.299,Z 853.502,A -85,B 0,C 180,E1 1358.791,E2 1358.791} C_VEL
LIN {X 0,Y 594.415,Z 836.722,A -85,B 0,C 180,E1 1362.315,E2 1362.315} C_VEL
LIN {X 0,Y 594.586,Z 815.278,A -85,B 0,C 180,E1 1365.506,E2 1365.506} C_VEL
LIN {X 0,Y 594.932,Z 788.599,A -85,B 0,C 180,E1 1368.451,E2 1368.451} C_VEL
LIN {X 0,Y 595.32,Z 757.694,A -85,B 0,C 180,E1 1370.977,E2 1370.977} C_VEL
LIN {X 0,Y 595.761,Z 724.855,A -85,B 0,C 180,E1 1372.947,E2 1372.947} C_VEL
LIN {X 0,Y 596.155,Z 688.531,A -85,B 0,C 180,E1 1374.45,E2 1374.45} C_VEL
LIN {X 0,Y 596.392,Z 654.535,A -85,B 0,C 180,E1 1375.302,E2 1375.302} C_VEL
LIN {X 0,Y 595.616,Z 587.108,A -85,B 0,C 180,E1 1376.25,E2 1376.25} C_VEL
LIN {X 0,Y 594.101,Z 580.66,A -85,B 0,C 180,E1 1376.443,E2 1376.443} C_VEL
LIN {X 0,Y 593.855,Z 580.66,A -85,B 0,C 180,E1 1382.727,E2 1382.727} C_VEL
LIN {X 0,Y 593.703,Z 580.66,A -85,B 0,C 180,E1 1387.77,E2 1387.77} C_VEL
LIN {X 0,Y 593.706,Z 580.66,A -85,B 0,C 180,E1 1393.512,E2 1393.512} C_VEL
LIN {X 0,Y 593.823,Z 580.66,A -85,B 0,C 180,E1 1398.484,E2 1398.484} C_VEL
LIN {X 0,Y 593.834,Z 580.66,A -85,B 0,C 180,E1 1404.67,E2 1404.67} C_VEL
LIN {X 0,Y 593.765,Z 580.66,A -85,B 0,C 180,E1 1411.026,E2 1411.026} C_VEL
LIN {X 0,Y 593.868,Z 580.66,A -85,B 0,C 180,E1 1415.931,E2 1415.931} C_VEL
LIN {X 0,Y 594.003,Z 580.66,A -85,B 0,C 180,E1 1420.654,E2 1420.654} C_VEL
LIN {X 0,Y 593.689,Z 580.66,A -85,B 0,C 180,E1 1425.229,E2 1425.229} C_VEL
LIN {X 0,Y 594.04,Z 580.66,A -85,B 0,C 180,E1 1429.727,E2 1429.727} C_VEL
LIN {X 0,Y 594.212,Z 580.66,A -85,B 0,C 180,E1 1434.154,E2 1434.154} C_VEL
LIN {X 0,Y 593.943,Z 580.66,A -85,B 0,C 180,E1 1440.004,E2 1440.004} C_VEL
LIN {X 0,Y 594.044,Z 580.66,A -85,B 0,C 180,E1 1444.389,E2 1444.389} C_VEL
LIN {X 0,Y 594.052,Z 580.66,A -85,B 0,C 180,E1 1448.8,E2 1448.8} C_VEL
LIN {X 0,Y 593.839,Z 580.66,A -85,B 0,C 180,E1 1454.349,E2 1454.349} C_VEL
LIN {X 0,Y 593.886,Z 580.66,A -85,B 0,C 180,E1 1459.398,E2 1459.398} C_VEL
LIN {X 0,Y 593.807,Z 580.66,A -85,B 0,C 180,E1 1464.081,E2 1464.081} C_VEL
LIN {X 0,Y 593.788,Z 580.66,A -85,B 0,C 180,E1 1468.982,E2 1468.982} C_VEL
LIN {X 0,Y 593.987,Z 580.66,A -85,B 0,C 180,E1 1474.114,E2 1474.114} C_VEL
LIN {X 0,Y 593.754,Z 580.66,A -85,B 0,C 180,E1 1480.098,E2 1480.098} C_VEL
LIN {X 0,Y 593.553,Z 580.66,A -85,B 0,C 180,E1 1485.585,E2 1485.585} C_VEL
LIN {X 0,Y 593.758,Z 580.66,A -85,B 0,C 180,E1 1490.398,E2 1490.398} C_VEL
LIN {X 0,Y 594.034,Z 580.66,A -85,B 0,C 180,E1 1495.896,E2 1495.896} C_VEL
LIN {X 0,Y 593.831,Z 580.66,A -85,B 0,C 180,E1 1501.027,E2 1501.027} C_VEL
LIN {X 0,Y 593.928,Z 580.66,A -85,B 0,C 180,E1 1507.521,E2 1507.521} C_VEL
LIN {X 0,Y 594.118,Z 580.933,A -85,B 0,C 180,E1 1510.309,E2 1510.309} C_VEL
LIN {X 0,Y 595.315,Z 597.999,A -85,B 0,C 180,E1 1511.081,E2 1511.081} C_VEL
LIN {X 0,Y 595.013,Z 629.073,A -85,B 0,C 180,E1 1512.9,E2 1512.9} C_VEL
LIN {X 0,Y 594.774,Z 655.318,A -85,B 0,C 180,E1 1515.066,E2 1515.066} C_VEL
LIN {X 0,Y 594.538,Z 678.491,A -85,B 0,C 180,E1 1517.687,E2 1517.687} C_VEL
LIN {X 0,Y 594.389,Z 696.095,A -85,B 0,C 180,E1 1520.471,E2 1520.471} C_VEL
LIN {X 0,Y 594.364,Z 709.886,A -85,B 0,C 180,E1 1523.698,E2 1523.698} C_VEL
LIN {X 0,Y 594.317,Z 717.884,A -85,B 0,C 180,E1 1527.081,E2 1527.081} C_VEL
LIN {X 0,Y 594.288,Z 719.996,A -85,B 0,C 180,E1 1530.001,E2 1530.001} C_VEL
LIN {X 0,Y 594.25,Z 717.733,A -85,B 0,C 180,E1 1532.922,E2 1532.922} C_VEL
LIN {X 0,Y 594.303,Z 709.774,A -85,B 0,C 180,E1 1536.248,E2 1536.248} C_VEL
LIN {X 0,Y 594.357,Z 697.56,A -85,B 0,C 180,E1 1539.162,E2 1539.162} C_VEL
LIN {X 0,Y 594.491,Z 679.167,A -85,B 0,C 180,E1 1542.13,E2 1542.13} C_VEL
LIN {X 0,Y 594.732,Z 656.289,A -85,B 0,C 180,E1 1544.75,E2 1544.75} C_VEL
LIN {X 0,Y 595.015,Z 628.819,A -85,B 0,C 180,E1 1547.027,E2 1547.027} C_VEL
LIN {X 0,Y 595.234,Z 598.071,A -85,B 0,C 180,E1 1548.829,E2 1548.829} C_VEL
LIN {X 0,Y 594.321,Z 580.66,A -85,B 0,C 180,E1 1549.609,E2 1549.609} C_VEL
LIN {X 0,Y 593.966,Z 580.66,A -85,B 0,C 180,E1 1555.681,E2 1555.681} C_VEL
LIN {X 0,Y 593.834,Z 580.66,A -85,B 0,C 180,E1 1560.66,E2 1560.66} C_VEL
LIN {X 0,Y 593.874,Z 580.66,A -85,B 0,C 180,E1 1565.901,E2 1565.901} C_VEL
LIN {X 0,Y 593.619,Z 580.66,A -85,B 0,C 180,E1 1571.541,E2 1571.541} C_VEL
LIN {X 0,Y 593.792,Z 580.66,A -85,B 0,C 180,E1 1576.488,E2 1576.488} C_VEL
LIN {X 0,Y 593.75,Z 580.66,A -85,B 0,C 180,E1 1582.262,E2 1582.262} C_VEL
LIN {X 0,Y 593.604,Z 580.66,A -85,B 0,C 180,E1 1587.609,E2 1587.609} C_VEL
LIN {X 0,Y 593.712,Z 580.66,A -85,B 0,C 180,E1 1592.672,E2 1592.672} C_VEL
LIN {X 0,Y 593.718,Z 580.66,A -85,B 0,C 180,E1 1597.506,E2 1597.506} C_VEL
LIN {X 0,Y 594.013,Z 580.66,A -85,B 0,C 180,E1 1602.186,E2 1602.186} C_VEL
LIN {X 0,Y 593.693,Z 580.66,A -85,B 0,C 180,E1 1608.224,E2 1608.224} C_VEL
LIN {X 0,Y 594.228,Z 580.66,A -85,B 0,C 180,E1 1614.146,E2 1614.146} C_VEL
LIN {X 0,Y 593.972,Z 580.66,A -85,B 0,C 180,E1 1619.996,E2 1619.996} C_VEL
LIN {X 0,Y 593.823,Z 580.66,A -85,B 0,C 180,E1 1621.114,E2 1621.114} C_VEL
LIN {X 0,Y 590.067,Z 580.66,A -85,B 0,C 180,E1 1622.769,E2 1622.769} C_VEL
LIN {X 0,Y 586.118,Z 580.66,A -85,B 0,C 180,E1 1624.444,E2 1624.444} C_VEL
LIN {X 0,Y 586.132,Z 580.66,A -85,B 0,C 180,E1 1628.912,E2 1628.912} C_VEL
LIN {X 0,Y 586.162,Z 580.66,A -85,B 0,C 180,E1 1633.438,E2 1633.438} C_VEL
LIN {X 0,Y 585.973,Z 580.66,A -85,B 0,C 180,E1 1639.622,E2 1639.622} C_VEL
LIN {X 0,Y 585.867,Z 580.66,A -85,B 0,C 180,E1 1644.419,E2 1644.419} C_VEL
LIN {X 0,Y 585.792,Z 580.66,A -85,B 0,C 180,E1 1649.406,E2 1649.406} C_VEL
LIN {X 0,Y 585.866,Z 580.66,A -85,B 0,C 180,E1 1654.643,E2 1654.643} C_VEL
LIN {X 0,Y 585.787,Z 580.66,A -85,B 0,C 180,E1 1660.247,E2 1660.247} C_VEL
LIN {X 0,Y 585.918,Z 580.66,A -85,B 0,C 180,E1 1666.34,E2 1666.34} C_VEL
LIN {X 0,Y 585.846,Z 580.66,A -85,B 0,C 180,E1 1671.665,E2 1671.665} C_VEL
LIN {X 0,Y 585.746,Z 580.66,A -85,B 0,C 180,E1 1677.124,E2 1677.124} C_VEL
LIN {X 0,Y 586.086,Z 580.66,A -85,B 0,C 180,E1 1683.16,E2 1683.16} C_VEL
LIN {X 0,Y 589.23,Z 593.183,A -85,B 0,C 180,E1 1683.524,E2 1683.524} C_VEL
LIN {X 0,Y 589.056,Z 666.19,A -85,B 0,C 180,E1 1684.602,E2 1684.602} C_VEL
LIN {X 0,Y 588.704,Z 703.019,A -85,B 0,C 180,E1 1685.758,E2 1685.758} C_VEL
LIN {X 0,Y 588.175,Z 736.678,A -85,B 0,C 180,E1 1687.392,E2 1687.392} C_VEL
LIN {X 0,Y 587.621,Z 768.738,A -85,B 0,C 180,E1 1689.57,E2 1689.57} C_VEL
LIN {X 0,Y 587.107,Z 798.959,A -85,B 0,C 180,E1 1692.358,E2 1692.358} C_VEL
LIN {X 0,Y 586.728,Z 822.97,A -85,B 0,C 180,E1 1695.331,E2 1695.331} C_VEL
LIN {X 0,Y 586.512,Z 842.058,A -85,B 0,C 180,E1 1698.514,E2 1698.514} C_VEL
LIN {X 0,Y 586.428,Z 856.172,A -85,B 0,C 180,E1 1701.835,E2 1701.835} C_VEL
LIN {X 0,Y 586.3,Z 865.967,A -85,B 0,C 180,E1 1705.555,E2 1705.555} C_VEL
LIN {X 0,Y 586.3,Z 869.507,A -85,B 0,C 180,E1 1708.519,E2 1708.519} C_VEL
LIN {X 0,Y 586.406,Z 869.509,A -85,B 0,C 180,E1 1711.478,E2 1711.478} C_VEL
LIN {X 0,Y 586.391,Z 864.456,A -85,B 0,C 180,E1 1715.183,E2 1715.183} C_VEL
LIN {X 0,Y 586.406,Z 853.502,A -85,B 0,C 180,E1 1718.91,E2 1718.91} C_VEL
LIN {X 0,Y 586.566,Z 837.81,A -85,B 0,C 180,E1 1722.294,E2 1722.294} C_VEL
LIN {X 0,Y 586.808,Z 816.747,A -85,B 0,C 180,E1 1725.525,E2 1725.525} C_VEL
LIN {X 0,Y 587.233,Z 791.519,A -85,B 0,C 180,E1 1728.41,E2 1728.41} C_VEL
LIN {X 0,Y 587.754,Z 761.395,A -85,B 0,C 180,E1 1730.995,E2 1730.995} C_VEL
LIN {X 0,Y 588.319,Z 727.919,A -85,B 0,C 180,E1 1733.091,E2 1733.091} C_VEL
LIN {X 0,Y 588.832,Z 693.575,A -85,B 0,C 180,E1 1734.594,E2 1734.594} C_VEL
LIN {X 0,Y 589.201,Z 657.445,A -85,B 0,C 180,E1 1735.574,E2 1735.574} C_VEL
LIN {X 0,Y 588.687,Z 589.243,A -85,B 0,C 180,E1 1736.555,E2 1736.555} C_VEL
LIN {X 0,Y 586.297,Z 580.66,A -85,B 0,C 180,E1 1736.838,E2 1736.838} C_VEL
LIN {X 0,Y 585.953,Z 580.66,A -85,B 0,C 180,E1 1742.86,E2 1742.86} C_VEL
LIN {X 0,Y 585.786,Z 580.66,A -85,B 0,C 180,E1 1749.167,E2 1749.167} C_VEL
LIN {X 0,Y 585.855,Z 580.66,A -85,B 0,C 180,E1 1754.245,E2 1754.245} C_VEL
LIN {X 0,Y 585.877,Z 580.66,A -85,B 0,C 180,E1 1759.761,E2 1759.761} C_VEL
LIN {X 0,Y 585.817,Z 580.66,A -85,B 0,C 180,E1 1765.354,E2 1765.354} C_VEL
LIN {X 0,Y 585.896,Z 580.66,A -85,B 0,C 180,E1 1770.599,E2 1770.599} C_VEL
LIN {X 0,Y 585.942,Z 580.66,A -85,B 0,C 180,E1 1775.584,E2 1775.584} C_VEL
LIN {X 0,Y 586.09,Z 580.66,A -85,B 0,C 180,E1 1780.382,E2 1780.382} C_VEL
LIN {X 0,Y 585.813,Z 580.66,A -85,B 0,C 180,E1 1785.026,E2 1785.026} C_VEL
LIN {X 0,Y 586.094,Z 580.66,A -85,B 0,C 180,E1 1789.586,E2 1789.586} C_VEL
LIN {X 0,Y 586.29,Z 580.66,A -85,B 0,C 180,E1 1794.075,E2 1794.075} C_VEL
LIN {X 0,Y 586.053,Z 580.66,A -85,B 0,C 180,E1 1800.004,E2 1800.004} C_VEL
LIN {X 0,Y 586.133,Z 580.66,A -85,B 0,C 180,E1 1804.449,E2 1804.449} C_VEL
LIN {X 0,Y 586.114,Z 580.66,A -85,B 0,C 180,E1 1808.92,E2 1808.92} C_VEL
LIN {X 0,Y 586.124,Z 580.66,A -85,B 0,C 180,E1 1813.447,E2 1813.447} C_VEL
LIN {X 0,Y 586.099,Z 580.66,A -85,B 0,C 180,E1 1818.063,E2 1818.063} C_VEL
LIN {X 0,Y 585.983,Z 580.66,A -85,B 0,C 180,E1 1822.807,E2 1822.807} C_VEL
LIN {X 0,Y 585.859,Z 580.66,A -85,B 0,C 180,E1 1828.523,E2 1828.523} C_VEL
LIN {X 0,Y 586.029,Z 580.66,A -85,B 0,C 180,E1 1834.642,E2 1834.642} C_VEL
LIN {X 0,Y 585.866,Z 580.66,A -85,B 0,C 180,E1 1840.251,E2 1840.251} C_VEL
LIN {X 0,Y 585.733,Z 580.66,A -85,B 0,C 180,E1 1846.371,E2 1846.371} C_VEL
LIN {X 0,Y 585.873,Z 580.66,A -85,B 0,C 180,E1 1851.67,E2 1851.67} C_VEL
LIN {X 0,Y 586.049,Z 580.66,A -85,B 0,C 180,E1 1857.146,E2 1857.146} C_VEL
LIN {X 0,Y 585.841,Z 580.66,A -85,B 0,C 180,E1 1862.279,E2 1862.279} C_VEL
LIN {X 0,Y 586.011,Z 580.66,A -85,B 0,C 180,E1 1868.462,E2 1868.462} C_VEL
LIN {X 0,Y 586.166,Z 580.854,A -85,B 0,C 180,E1 1870.029,E2 1870.029} C_VEL
LIN {X 0,Y 587.779,Z 594.832,A -85,B 0,C 180,E1 1870.682,E2 1870.682} C_VEL
LIN {X 0,Y 587.425,Z 626.586,A -85,B 0,C 180,E1 1872.498,E2 1872.498} C_VEL
LIN {X 0,Y 587.024,Z 653.382,A -85,B 0,C 180,E1 1874.672,E2 1874.672} C_VEL
LIN {X 0,Y 586.737,Z 677.041,A -85,B 0,C 180,E1 1877.331,E2 1877.331} C_VEL
LIN {X 0,Y 586.519,Z 696.092,A -85,B 0,C 180,E1 1880.342,E2 1880.342} C_VEL
LIN {X 0,Y 586.443,Z 709.224,A -85,B 0,C 180,E1 1883.408,E2 1883.408} C_VEL
LIN {X 0,Y 586.399,Z 716.689,A -85,B 0,C 180,E1 1886.301,E2 1886.301} C_VEL
LIN {X 0,Y 586.347,Z 719.449,A -85,B 0,C 180,E1 1888.522,E2 1888.522} C_VEL
LIN {X 0,Y 586.358,Z 719.385,A -85,B 0,C 180,E1 1891.481,E2 1891.481} C_VEL
LIN {X 0,Y 586.406,Z 714.974,A -85,B 0,C 180,E1 1894.444,E2 1894.444} C_VEL
LIN {X 0,Y 586.458,Z 704.372,A -85,B 0,C 180,E1 1897.791,E2 1897.791} C_VEL
LIN {X 0,Y 586.579,Z 689.054,A -85,B 0,C 180,E1 1900.82,E2 1900.82} C_VEL
LIN {X 0,Y 586.834,Z 667.613,A -85,B 0,C 180,E1 1903.743,E2 1903.743} C_VEL
LIN {X 0,Y 587.214,Z 641.511,A -85,B 0,C 180,E1 1906.285,E2 1906.285} C_VEL
LIN {X 0,Y 587.606,Z 612.54,A -85,B 0,C 180,E1 1908.303,E2 1908.303} C_VEL
LIN {X 0,Y 586.962,Z 583.603,A -85,B 0,C 180,E1 1909.742,E2 1909.742} C_VEL
LIN {X 0,Y 586.324,Z 580.66,A -85,B 0,C 180,E1 1909.968,E2 1909.968} C_VEL
LIN {X 0,Y 586.006,Z 580.66,A -85,B 0,C 180,E1 1916.055,E2 1916.055} C_VEL
LIN {X 0,Y 585.797,Z 580.66,A -85,B 0,C 180,E1 1921.463,E2 1921.463} C_VEL
LIN {X 0,Y 585.947,Z 580.66,A -85,B 0,C 180,E1 1926.767,E2 1926.767} C_VEL
LIN {X 0,Y 585.723,Z 580.66,A -85,B 0,C 180,E1 1932.229,E2 1932.229} C_VEL
LIN {X 0,Y 585.889,Z 580.66,A -85,B 0,C 180,E1 1937.782,E2 1937.782} C_VEL
LIN {X 0,Y 585.827,Z 580.66,A -85,B 0,C 180,E1 1943.524,E2 1943.524} C_VEL
LIN {X 0,Y 585.788,Z 580.66,A -85,B 0,C 180,E1 1948.869,E2 1948.869} C_VEL
LIN {X 0,Y 586.003,Z 580.66,A -85,B 0,C 180,E1 1954.729,E2 1954.729} C_VEL
LIN {X 0,Y 586.122,Z 580.66,A -85,B 0,C 180,E1 1960.374,E2 1960.374} C_VEL
LIN {X 0,Y 585.797,Z 580.66,A -85,B 0,C 180,E1 1965.017,E2 1965.017} C_VEL
LIN {X 0,Y 585.923,Z 580.66,A -85,B 0,C 180,E1 1971.077,E2 1971.077} C_VEL
LIN {X 0,Y 586.021,Z 580.66,A -85,B 0,C 180,E1 1975.551,E2 1975.551} C_VEL
LIN {X 0,Y 586.082,Z 580.66,A -85,B 0,C 180,E1 1979.996,E2 1979.996} C_VEL
LIN {X 0,Y 586.118,Z 580.66,A -85,B 0,C 180,E1 1984.444,E2 1984.444} C_VEL
LIN {X 0,Y 582.063,Z 580.66,A -85,B 0,C 180,E1 1986.11,E2 1986.11} C_VEL
LIN {X 0,Y 578.145,Z 580.66,A -85,B 0,C 180,E1 1987.799,E2 1987.799} C_VEL
LIN {X 0,Y 578.201,Z 580.66,A -85,B 0,C 180,E1 1993.627,E2 1993.627} C_VEL
LIN {X 0,Y 578.084,Z 580.66,A -85,B 0,C 180,E1 1999.46,E2 1999.46} C_VEL
LIN {X 0,Y 577.959,Z 580.66,A -85,B 0,C 180,E1 2004.776,E2 2004.776} C_VEL
LIN {X 0,Y 577.824,Z 580.66,A -85,B 0,C 180,E1 2010.152,E2 2010.152} C_VEL
LIN {X 0,Y 577.848,Z 580.66,A -85,B 0,C 180,E1 2015.194,E2 2015.194} C_VEL
LIN {X 0,Y 577.83,Z 580.66,A -85,B 0,C 180,E1 2020.918,E2 2020.918} C_VEL
LIN {X 0,Y 577.984,Z 580.66,A -85,B 0,C 180,E1 2027.171,E2 2027.171} C_VEL
LIN {X 0,Y 577.966,Z 580.66,A -85,B 0,C 180,E1 2032.949,E2 2032.949} C_VEL
LIN {X 0,Y 577.92,Z 580.66,A -85,B 0,C 180,E1 2038.401,E2 2038.401} C_VEL
LIN {X 0,Y 578.138,Z 580.765,A -85,B 0,C 180,E1 2042.806,E2 2042.806} C_VEL
LIN {X 0,Y 582.173,Z 595.651,A -85,B 0,C 180,E1 2043.211,E2 2043.211} C_VEL
LIN {X 0,Y 581.914,Z 666.498,A -85,B 0,C 180,E1 2044.275,E2 2044.275} C_VEL
LIN {X 0,Y 581.449,Z 703.253,A -85,B 0,C 180,E1 2045.446,E2 2045.446} C_VEL
LIN {X 0,Y 580.751,Z 736.679,A -85,B 0,C 180,E1 2047.086,E2 2047.086} C_VEL
LIN {X 0,Y 580.079,Z 768.44,A -85,B 0,C 180,E1 2049.268,E2 2049.268} C_VEL
LIN {X 0,Y 579.479,Z 797.207,A -85,B 0,C 180,E1 2051.922,E2 2051.922} C_VEL
LIN {X 0,Y 578.953,Z 822.133,A -85,B 0,C 180,E1 2055.008,E2 2055.008} C_VEL
LIN {X 0,Y 578.664,Z 841.651,A -85,B 0,C 180,E1 2058.276,E2 2058.276} C_VEL
LIN {X 0,Y 578.549,Z 856.172,A -85,B 0,C 180,E1 2061.723,E2 2061.723} C_VEL
LIN {X 0,Y 578.405,Z 865.966,A -85,B 0,C 180,E1 2065.495,E2 2065.495} C_VEL
LIN {X 0,Y 578.4,Z 869.507,A -85,B 0,C 180,E1 2068.499,E2 2068.499} C_VEL
LIN {X 0,Y 578.501,Z 869.509,A -85,B 0,C 180,E1 2071.498,E2 2071.498} C_VEL
LIN {X 0,Y 578.501,Z 864.49,A -85,B 0,C 180,E1 2075.238,E2 2075.238} C_VEL
LIN {X 0,Y 578.523,Z 853.502,A -85,B 0,C 180,E1 2079.033,E2 2079.033} C_VEL
LIN {X 0,Y 578.713,Z 837.809,A -85,B 0,C 180,E1 2082.463,E2 2082.463} C_VEL
LIN {X 0,Y 579.046,Z 816.749,A -85,B 0,C 180,E1 2085.739,E2 2085.739} C_VEL
LIN {X 0,Y 579.561,Z 791.518,A -85,B 0,C 180,E1 2088.662,E2 2088.662} C_VEL
LIN {X 0,Y 580.232,Z 760.921,A -85,B 0,C 180,E1 2091.315,E2 2091.315} C_VEL
LIN {X 0,Y 580.988,Z 727.77,A -85,B 0,C 180,E1 2093.408,E2 2093.408} C_VEL
LIN {X 0,Y 581.615,Z 693.459,A -85,B 0,C 180,E1 2094.925,E2 2094.925} C_VEL
LIN {X 0,Y 582.107,Z 656.272,A -85,B 0,C 180,E1 2095.933,E2 2095.933} C_VEL
LIN {X 0,Y 581.719,Z 591.085,A -85,B 0,C 180,E1 2096.873,E2 2096.873} C_VEL
LIN {X 0,Y 578.316,Z 580.66,A -85,B 0,C 180,E1 2097.247,E2 2097.247} C_VEL
LIN {X 0,Y 578.03,Z 580.66,A -85,B 0,C 180,E1 2103.369,E2 2103.369} C_VEL
LIN {X 0,Y 577.871,Z 580.66,A -85,B 0,C 180,E1 2108.96,E2 2108.96} C_VEL
LIN {X 0,Y 577.947,Z 580.66,A -85,B 0,C 180,E1 2115.014,E2 2115.014} C_VEL
LIN {X 0,Y 577.978,Z 580.66,A -85,B 0,C 180,E1 2119.432,E2 2119.432} C_VEL
LIN {X 0,Y 577.87,Z 580.66,A -85,B 0,C 180,E1 2124.807,E2 2124.807} C_VEL
LIN {X 0,Y 577.935,Z 580.66,A -85,B 0,C 180,E1 2130.154,E2 2130.154} C_VEL
LIN {X 0,Y 578.064,Z 580.66,A -85,B 0,C 180,E1 2135.229,E2 2135.229} C_VEL
LIN {X 0,Y 578.175,Z 580.66,A -85,B 0,C 180,E1 2140.506,E2 2140.506} C_VEL
LIN {X 0,Y 577.929,Z 580.66,A -85,B 0,C 180,E1 2144.817,E2 2144.817} C_VEL
LIN {X 0,Y 578.038,Z 580.66,A -85,B 0,C 180,E1 2150.962,E2 2150.962} C_VEL
LIN {X 0,Y 578.09,Z 580.66,A -85,B 0,C 180,E1 2155.498,E2 2155.498} C_VEL
LIN {X 0,Y 578.153,Z 580.66,A -85,B 0,C 180,E1 2160.004,E2 2160.004} C_VEL
LIN {X 0,Y 578.218,Z 580.66,A -85,B 0,C 180,E1 2164.51,E2 2164.51} C_VEL
LIN {X 0,Y 578.179,Z 580.66,A -85,B 0,C 180,E1 2169.044,E2 2169.044} C_VEL
LIN {X 0,Y 578.031,Z 580.66,A -85,B 0,C 180,E1 2174.279,E2 2174.279} C_VEL
LIN {X 0,Y 578.045,Z 580.66,A -85,B 0,C 180,E1 2179.912,E2 2179.912} C_VEL
LIN {X 0,Y 577.943,Z 580.66,A -85,B 0,C 180,E1 2184.786,E2 2184.786} C_VEL
LIN {X 0,Y 577.868,Z 580.66,A -85,B 0,C 180,E1 2190.165,E2 2190.165} C_VEL
LIN {X 0,Y 578.022,Z 580.66,A -85,B 0,C 180,E1 2195.192,E2 2195.192} C_VEL
LIN {X 0,Y 577.932,Z 580.66,A -85,B 0,C 180,E1 2200.92,E2 2200.92} C_VEL
LIN {X 0,Y 577.86,Z 580.66,A -85,B 0,C 180,E1 2207.197,E2 2207.197} C_VEL
LIN {X 0,Y 578.01,Z 580.66,A -85,B 0,C 180,E1 2212.956,E2 2212.956} C_VEL
LIN {X 0,Y 578.026,Z 580.66,A -85,B 0,C 180,E1 2218.41,E2 2218.41} C_VEL
LIN {X 0,Y 577.881,Z 580.66,A -85,B 0,C 180,E1 2223.553,E2 2223.553} C_VEL
LIN {X 0,Y 578.215,Z 580.66,A -85,B 0,C 180,E1 2229.702,E2 2229.702} C_VEL
LIN {X 0,Y 580.268,Z 594.948,A -85,B 0,C 180,E1 2230.428,E2 2230.428} C_VEL
LIN {X 0,Y 579.802,Z 626.572,A -85,B 0,C 180,E1 2232.261,E2 2232.261} C_VEL
LIN {X 0,Y 579.337,Z 653.375,A -85,B 0,C 180,E1 2234.464,E2 2234.464} C_VEL
LIN {X 0,Y 578.904,Z 677.035,A -85,B 0,C 180,E1 2237.157,E2 2237.157} C_VEL
LIN {X 0,Y 578.657,Z 696.09,A -85,B 0,C 180,E1 2240.21,E2 2240.21} C_VEL
LIN {X 0,Y 578.561,Z 708.946,A -85,B 0,C 180,E1 2243.239,E2 2243.239} C_VEL
LIN {X 0,Y 578.515,Z 716.687,A -85,B 0,C 180,E1 2246.25,E2 2246.25} C_VEL
LIN {X 0,Y 578.446,Z 719.449,A -85,B 0,C 180,E1 2248.502,E2 2248.502} C_VEL
LIN {X 0,Y 578.455,Z 719.386,A -85,B 0,C 180,E1 2251.501,E2 2251.501} C_VEL
LIN {X 0,Y 578.503,Z 714.974,A -85,B 0,C 180,E1 2254.505,E2 2254.505} C_VEL
LIN {X 0,Y 578.588,Z 704.375,A -85,B 0,C 180,E1 2257.898,E2 2257.898} C_VEL
LIN {X 0,Y 578.754,Z 687.982,A -85,B 0,C 180,E1 2261.139,E2 2261.139} C_VEL
LIN {X 0,Y 579.073,Z 666.916,A -85,B 0,C 180,E1 2264.016,E2 2264.016} C_VEL
LIN {X 0,Y 579.534,Z 640.366,A -85,B 0,C 180,E1 2266.605,E2 2266.605} C_VEL
LIN {X 0,Y 580.068,Z 610.864,A -85,B 0,C 180,E1 2268.648,E2 2268.648} C_VEL
LIN {X 0,Y 579.338,Z 585.112,A -85,B 0,C 180,E1 2269.952,E2 2269.952} C_VEL
LIN {X 0,Y 578.364,Z 580.66,A -85,B 0,C 180,E1 2270.256,E2 2270.256} C_VEL
LIN {X 0,Y 578.013,Z 580.66,A -85,B 0,C 180,E1 2276.443,E2 2276.443} C_VEL
LIN {X 0,Y 577.891,Z 580.66,A -85,B 0,C 180,E1 2281.601,E2 2281.601} C_VEL
LIN {X 0,Y 578.035,Z 580.66,A -85,B 0,C 180,E1 2287.046,E2 2287.046} C_VEL
LIN {X 0,Y 577.845,Z 580.66,A -85,B 0,C 180,E1 2292.942,E2 2292.942} C_VEL
LIN {X 0,Y 577.975,Z 580.66,A -85,B 0,C 180,E1 2297.18,E2 2297.18} C_VEL
LIN {X 0,Y 577.914,Z 580.66,A -85,B 0,C 180,E1 2302.941,E2 2302.941} C_VEL
LIN {X 0,Y 577.859,Z 580.66,A -85,B 0,C 180,E1 2308.393,E2 2308.393} C_VEL
LIN {X 0,Y 577.989,Z 580.66,A -85,B 0,C 180,E1 2313.552,E2 2313.552} C_VEL
LIN {X 0,Y 578.054,Z 580.66,A -85,B 0,C 180,E1 2318.484,E2 2318.484} C_VEL
LIN {X 0,Y 578.197,Z 580.66,A -85,B 0,C 180,E1 2323.255,E2 2323.255} C_VEL
LIN {X 0,Y 578.131,Z 580.66,A -85,B 0,C 180,E1 2329.433,E2 2329.433} C_VEL
LIN {X 0,Y 578.39,Z 580.66,A -85,B 0,C 180,E1 2334.114,E2 2334.114} C_VEL
LIN {X 0,Y 578.181,Z 580.66,A -85,B 0,C 180,E1 2339.996,E2 2339.996} C_VEL
LIN {X 0,Y 578.203,Z 580.66,A -85,B 0,C 180,E1 2344.501,E2 2344.501} C_VEL
LIN {X 0,Y 578.145,Z 580.66,A -85,B 0,C 180,E1 2347.799,E2 2347.799} C_VEL
LIN {X 0,Y 576.843,Z 580.66,A -85,B 0,C 180,E1 2348.654,E2 2348.654} C_VEL
LIN {X 0,Y 570.205,Z 580.66,A -85,B 0,C 180,E1 2350.981,E2 2350.981} C_VEL
LIN {X 0,Y 570.116,Z 580.66,A -85,B 0,C 180,E1 2351.201,E2 2351.201} C_VEL
LIN {X 0,Y 570.077,Z 580.66,A -85,B 0,C 180,E1 2355.397,E2 2355.397} C_VEL
LIN {X 0,Y 570.107,Z 580.66,A -85,B 0,C 180,E1 2360.192,E2 2360.192} C_VEL
LIN {X 0,Y 570.006,Z 580.66,A -85,B 0,C 180,E1 2365.43,E2 2365.43} C_VEL
LIN {X 0,Y 569.941,Z 580.66,A -85,B 0,C 180,E1 2370.308,E2 2370.308} C_VEL
LIN {X 0,Y 569.909,Z 580.66,A -85,B 0,C 180,E1 2375.759,E2 2375.759} C_VEL
LIN {X 0,Y 569.868,Z 580.66,A -85,B 0,C 180,E1 2381.615,E2 2381.615} C_VEL
LIN {X 0,Y 569.98,Z 580.66,A -85,B 0,C 180,E1 2386.318,E2 2386.318} C_VEL
LIN {X 0,Y 570.046,Z 580.66,A -85,B 0,C 180,E1 2392.346,E2 2392.346} C_VEL
LIN {X 0,Y 570.001,Z 580.66,A -85,B 0,C 180,E1 2398.201,E2 2398.201} C_VEL
LIN {X 0,Y 570.172,Z 580.66,A -85,B 0,C 180,E1 2402.392,E2 2402.392} C_VEL
LIN {X 0,Y 575.099,Z 595.686,A -85,B 0,C 180,E1 2402.855,E2 2402.855} C_VEL
LIN {X 0,Y 574.776,Z 667.181,A -85,B 0,C 180,E1 2403.95,E2 2403.95} C_VEL
LIN {X 0,Y 574.18,Z 704.063,A -85,B 0,C 180,E1 2405.149,E2 2405.149} C_VEL
LIN {X 0,Y 573.336,Z 738.407,A -85,B 0,C 180,E1 2406.878,E2 2406.878} C_VEL
LIN {X 0,Y 572.495,Z 770.935,A -85,B 0,C 180,E1 2409.183,E2 2409.183} C_VEL
LIN {X 0,Y 571.712,Z 800.539,A -85,B 0,C 180,E1 2412.046,E2 2412.046} C_VEL
LIN {X 0,Y 571.121,Z 824.605,A -85,B 0,C 180,E1 2415.162,E2 2415.162} C_VEL
LIN {X 0,Y 570.803,Z 843.243,A -85,B 0,C 180,E1 2418.429,E2 2418.429} C_VEL
LIN {X 0,Y 570.636,Z 857.455,A -85,B 0,C 180,E1 2421.992,E2 2421.992} C_VEL
LIN {X 0,Y 570.537,Z 865.966,A -85,B 0,C 180,E1 2425.432,E2 2425.432} C_VEL
LIN {X 0,Y 570.508,Z 869.507,A -85,B 0,C 180,E1 2428.478,E2 2428.478} C_VEL
LIN {X 0,Y 570.601,Z 869.509,A -85,B 0,C 180,E1 2431.519,E2 2431.519} C_VEL
LIN {X 0,Y 570.621,Z 864.751,A -85,B 0,C 180,E1 2435.182,E2 2435.182} C_VEL
LIN {X 0,Y 570.663,Z 854.842,A -85,B 0,C 180,E1 2438.773,E2 2438.773} C_VEL
LIN {X 0,Y 570.864,Z 838.843,A -85,B 0,C 180,E1 2442.443,E2 2442.443} C_VEL
LIN {X 0,Y 571.252,Z 818.208,A -85,B 0,C 180,E1 2445.762,E2 2445.762} C_VEL
LIN {X 0,Y 571.88,Z 793.479,A -85,B 0,C 180,E1 2448.717,E2 2448.717} C_VEL
LIN {X 0,Y 572.685,Z 763.439,A -85,B 0,C 180,E1 2451.416,E2 2451.416} C_VEL
LIN {X 0,Y 573.623,Z 729.075,A -85,B 0,C 180,E1 2453.656,E2 2453.656} C_VEL
LIN {X 0,Y 574.397,Z 693.982,A -85,B 0,C 180,E1 2455.24,E2 2455.24} C_VEL
LIN {X 0,Y 574.946,Z 658.614,A -85,B 0,C 180,E1 2456.23,E2 2456.23} C_VEL
LIN {X 0,Y 574.404,Z 591.906,A -85,B 0,C 180,E1 2457.232,E2 2457.232} C_VEL
LIN {X 0,Y 570.342,Z 580.66,A -85,B 0,C 180,E1 2457.637,E2 2457.637} C_VEL
LIN {X 0,Y 570.021,Z 580.66,A -85,B 0,C 180,E1 2463.9,E2 2463.9} C_VEL
LIN {X 0,Y 569.933,Z 580.66,A -85,B 0,C 180,E1 2469.618,E2 2469.618} C_VEL
LIN {X 0,Y 569.981,Z 580.66,A -85,B 0,C 180,E1 2475.821,E2 2475.821} C_VEL
LIN {X 0,Y 569.993,Z 580.66,A -85,B 0,C 180,E1 2480.4,E2 2480.4} C_VEL
LIN {X 0,Y 569.907,Z 580.66,A -85,B 0,C 180,E1 2485.439,E2 2485.439} C_VEL
LIN {X 0,Y 569.975,Z 580.66,A -85,B 0,C 180,E1 2491.229,E2 2491.229} C_VEL
LIN {X 0,Y 570.064,Z 580.66,A -85,B 0,C 180,E1 2496.527,E2 2496.527} C_VEL
LIN {X 0,Y 570.248,Z 580.66,A -85,B 0,C 180,E1 2501.426,E2 2501.426} C_VEL
LIN {X 0,Y 569.866,Z 580.66,A -85,B 0,C 180,E1 2506.17,E2 2506.17} C_VEL
LIN {X 0,Y 570.134,Z 580.66,A -85,B 0,C 180,E1 2510.836,E2 2510.836} C_VEL
LIN {X 0,Y 570.211,Z 580.66,A -85,B 0,C 180,E1 2515.435,E2 2515.435} C_VEL
LIN {X 0,Y 570.266,Z 580.66,A -85,B 0,C 180,E1 2520.004,E2 2520.004} C_VEL
LIN {X 0,Y 570.315,Z 580.66,A -85,B 0,C 180,E1 2524.572,E2 2524.572} C_VEL
LIN {X 0,Y 570.248,Z 580.66,A -85,B 0,C 180,E1 2529.171,E2 2529.171} C_VEL
LIN {X 0,Y 570.231,Z 580.66,A -85,B 0,C 180,E1 2533.83,E2 2533.83} C_VEL
LIN {X 0,Y 570.219,Z 580.66,A -85,B 0,C 180,E1 2538.584,E2 2538.584} C_VEL
LIN {X 0,Y 570.114,Z 580.66,A -85,B 0,C 180,E1 2543.48,E2 2543.48} C_VEL
LIN {X 0,Y 570.004,Z 580.66,A -85,B 0,C 180,E1 2548.776,E2 2548.776} C_VEL
LIN {X 0,Y 570.117,Z 580.66,A -85,B 0,C 180,E1 2554.592,E2 2554.592} C_VEL
LIN {X 0,Y 569.99,Z 580.66,A -85,B 0,C 180,E1 2559.621,E2 2559.621} C_VEL
LIN {X 0,Y 569.788,Z 580.66,A -85,B 0,C 180,E1 2565.849,E2 2565.849} C_VEL
LIN {X 0,Y 569.999,Z 580.66,A -85,B 0,C 180,E1 2570.397,E2 2570.397} C_VEL
LIN {X 0,Y 570.163,Z 580.66,A -85,B 0,C 180,E1 2576.109,E2 2576.109} C_VEL
LIN {X 0,Y 570.013,Z 580.66,A -85,B 0,C 180,E1 2581.44,E2 2581.44} C_VEL
LIN {X 0,Y 570.126,Z 580.66,A -85,B 0,C 180,E1 2586.527,E2 2586.527} C_VEL
LIN {X 0,Y 570.296,Z 580.765,A -85,B 0,C 180,E1 2589.446,E2 2589.446} C_VEL
LIN {X 0,Y 572.758,Z 594.938,A -85,B 0,C 180,E1 2590.16,E2 2590.16} C_VEL
LIN {X 0,Y 572.222,Z 626.284,A -85,B 0,C 180,E1 2591.998,E2 2591.998} C_VEL
LIN {X 0,Y 571.6,Z 653.367,A -85,B 0,C 180,E1 2594.248,E2 2594.248} C_VEL
LIN {X 0,Y 571.099,Z 677.029,A -85,B 0,C 180,E1 2596.979,E2 2596.979} C_VEL
LIN {X 0,Y 570.779,Z 696.088,A -85,B 0,C 180,E1 2600.073,E2 2600.073} C_VEL
LIN {X 0,Y 570.664,Z 708.942,A -85,B 0,C 180,E1 2603.145,E2 2603.145} C_VEL
LIN {X 0,Y 570.609,Z 716.685,A -85,B 0,C 180,E1 2606.198,E2 2606.198} C_VEL
LIN {X 0,Y 570.557,Z 719.449,A -85,B 0,C 180,E1 2608.481,E2 2608.481} C_VEL
LIN {X 0,Y 570.565,Z 719.385,A -85,B 0,C 180,E1 2611.522,E2 2611.522} C_VEL
LIN {X 0,Y 570.627,Z 714.975,A -85,B 0,C 180,E1 2614.567,E2 2614.567} C_VEL
LIN {X 0,Y 570.725,Z 704.377,A -85,B 0,C 180,E1 2618.007,E2 2618.007} C_VEL
LIN {X 0,Y 570.903,Z 688.252,A -85,B 0,C 180,E1 2621.251,E2 2621.251} C_VEL
LIN {X 0,Y 571.323,Z 666.433,A -85,B 0,C 180,E1 2624.268,E2 2624.268} C_VEL
LIN {X 0,Y 571.86,Z 640.371,A -85,B 0,C 180,E1 2626.834,E2 2626.834} C_VEL
LIN {X 0,Y 572.517,Z 610.665,A -85,B 0,C 180,E1 2628.916,E2 2628.916} C_VEL
LIN {X 0,Y 571.958,Z 587.3,A -85,B 0,C 180,E1 2630.13,E2 2630.13} C_VEL
LIN {X 0,Y 570.374,Z 580.66,A -85,B 0,C 180,E1 2630.549,E2 2630.549} C_VEL
LIN {X 0,Y 570.076,Z 580.66,A -85,B 0,C 180,E1 2636.841,E2 2636.841} C_VEL
LIN {X 0,Y 569.942,Z 580.66,A -85,B 0,C 180,E1 2642.094,E2 2642.094} C_VEL
LIN {X 0,Y 570.13,Z 580.66,A -85,B 0,C 180,E1 2647.648,E2 2647.648} C_VEL
LIN {X 0,Y 569.911,Z 580.66,A -85,B 0,C 180,E1 2654.163,E2 2654.163} C_VEL
LIN {X 0,Y 569.969,Z 580.66,A -85,B 0,C 180,E1 2658.382,E2 2658.382} C_VEL
LIN {X 0,Y 569.961,Z 580.66,A -85,B 0,C 180,E1 2664.234,E2 2664.234} C_VEL
LIN {X 0,Y 569.983,Z 580.66,A -85,B 0,C 180,E1 2669.684,E2 2669.684} C_VEL
LIN {X 0,Y 570.124,Z 580.66,A -85,B 0,C 180,E1 2674.851,E2 2674.851} C_VEL
LIN {X 0,Y 570.222,Z 580.66,A -85,B 0,C 180,E1 2679.803,E2 2679.803} C_VEL
LIN {X 0,Y 570.033,Z 580.66,A -85,B 0,C 180,E1 2684.593,E2 2684.593} C_VEL
LIN {X 0,Y 570.126,Z 580.66,A -85,B 0,C 180,E1 2690.827,E2 2690.827} C_VEL
LIN {X 0,Y 570.247,Z 580.66,A -85,B 0,C 180,E1 2695.427,E2 2695.427} C_VEL
LIN {X 0,Y 570.294,Z 580.66,A -85,B 0,C 180,E1 2699.996,E2 2699.996} C_VEL
LIN {X 0,Y 570.301,Z 580.66,A -85,B 0,C 180,E1 2704.564,E2 2704.564} C_VEL
LIN {X 0,Y 570.267,Z 580.66,A -85,B 0,C 180,E1 2709.162,E2 2709.162} C_VEL
LIN {X 0,Y 570.116,Z 580.66,A -85,B 0,C 180,E1 2711.201,E2 2711.201} C_VEL
LIN {X 0,Y 568.896,Z 580.66,A -85,B 0,C 180,E1 2712.069,E2 2712.069} C_VEL
LIN {X 0,Y 562.209,Z 580.66,A -85,B 0,C 180,E1 2714.654,E2 2714.654} C_VEL
LIN {X 0,Y 562.204,Z 580.66,A -85,B 0,C 180,E1 2720.488,E2 2720.488} C_VEL
LIN {X 0,Y 562.11,Z 580.66,A -85,B 0,C 180,E1 2725.523,E2 2725.523} C_VEL
LIN {X 0,Y 562.024,Z 580.66,A -85,B 0,C 180,E1 2730.781,E2 2730.781} C_VEL
LIN {X 0,Y 561.993,Z 580.66,A -85,B 0,C 180,E1 2736.343,E2 2736.343} C_VEL
LIN {X 0,Y 561.946,Z 580.66,A -85,B 0,C 180,E1 2742.337,E2 2742.337} C_VEL
LIN {X 0,Y 562.059,Z 580.66,A -85,B 0,C 180,E1 2747.666,E2 2747.666} C_VEL
LIN {X 0,Y 562.101,Z 580.66,A -85,B 0,C 180,E1 2753.899,E2 2753.899} C_VEL
LIN {X 0,Y 562.141,Z 580.66,A -85,B 0,C 180,E1 2759.518,E2 2759.518} C_VEL
LIN {X 0,Y 562.24,Z 580.66,A -85,B 0,C 180,E1 2761.947,E2 2761.947} C_VEL
LIN {X 0,Y 568.117,Z 598.476,A -85,B 0,C 180,E1 2762.533,E2 2762.533} C_VEL
LIN {X 0,Y 567.664,Z 667.514,A -85,B 0,C 180,E1 2763.607,E2 2763.607} C_VEL
LIN {X 0,Y 566.95,Z 703.886,A -85,B 0,C 180,E1 2764.803,E2 2764.803} C_VEL
LIN {X 0,Y 565.963,Z 738.802,A -85,B 0,C 180,E1 2766.583,E2 2766.583} C_VEL
LIN {X 0,Y 564.947,Z 772.139,A -85,B 0,C 180,E1 2768.994,E2 2768.994} C_VEL
LIN {X 0,Y 564.015,Z 800.938,A -85,B 0,C 180,E1 2771.838,E2 2771.838} C_VEL
LIN {X 0,Y 563.363,Z 824.668,A -85,B 0,C 180,E1 2774.963,E2 2774.963} C_VEL
LIN {X 0,Y 562.938,Z 843.715,A -85,B 0,C 180,E1 2778.361,E2 2778.361} C_VEL
LIN {X 0,Y 562.763,Z 857.455,A -85,B 0,C 180,E1 2781.879,E2 2781.879} C_VEL
LIN {X 0,Y 562.644,Z 865.965,A -85,B 0,C 180,E1 2785.368,E2 2785.368} C_VEL
LIN {X 0,Y 562.607,Z 869.508,A -85,B 0,C 180,E1 2788.457,E2 2788.457} C_VEL
LIN {X 0,Y 562.697,Z 869.51,A -85,B 0,C 180,E1 2791.54,E2 2791.54} C_VEL
LIN {X 0,Y 562.683,Z 864.38,A -85,B 0,C 180,E1 2795.441,E2 2795.441} C_VEL
LIN {X 0,Y 562.778,Z 853.502,A -85,B 0,C 180,E1 2799.288,E2 2799.288} C_VEL
LIN {X 0,Y 563.047,Z 837.808,A -85,B 0,C 180,E1 2802.816,E2 2802.816} C_VEL
LIN {X 0,Y 563.504,Z 816.749,A -85,B 0,C 180,E1 2806.184,E2 2806.184} C_VEL
LIN {X 0,Y 564.321,Z 790.241,A -85,B 0,C 180,E1 2809.321,E2 2809.321} C_VEL
LIN {X 0,Y 565.348,Z 759.414,A -85,B 0,C 180,E1 2812.018,E2 2812.018} C_VEL
LIN {X 0,Y 566.351,Z 726.639,A -85,B 0,C 180,E1 2814.114,E2 2814.114} C_VEL
LIN {X 0,Y 567.287,Z 692.079,A -85,B 0,C 180,E1 2815.651,E2 2815.651} C_VEL
LIN {X 0,Y 567.973,Z 655.127,A -85,B 0,C 180,E1 2816.653,E2 2816.653} C_VEL
LIN {X 0,Y 567.528,Z 594.402,A -85,B 0,C 180,E1 2817.555,E2 2817.555} C_VEL
LIN {X 0,Y 562.335,Z 580.66,A -85,B 0,C 180,E1 2818.086,E2 2818.086} C_VEL
LIN {X 0,Y 562.093,Z 580.66,A -85,B 0,C 180,E1 2824.445,E2 2824.445} C_VEL
LIN {X 0,Y 561.958,Z 580.66,A -85,B 0,C 180,E1 2830.284,E2 2830.284} C_VEL
LIN {X 0,Y 562.065,Z 580.66,A -85,B 0,C 180,E1 2835.55,E2 2835.55} C_VEL
LIN {X 0,Y 562.051,Z 580.66,A -85,B 0,C 180,E1 2841.721,E2 2841.721} C_VEL
LIN {X 0,Y 561.983,Z 580.66,A -85,B 0,C 180,E1 2847.402,E2 2847.402} C_VEL
LIN {X 0,Y 562.095,Z 580.66,A -85,B 0,C 180,E1 2852.753,E2 2852.753} C_VEL
LIN {X 0,Y 562.146,Z 580.66,A -85,B 0,C 180,E1 2857.853,E2 2857.853} C_VEL
LIN {X 0,Y 562.36,Z 580.66,A -85,B 0,C 180,E1 2862.778,E2 2862.778} C_VEL
LIN {X 0,Y 562.302,Z 580.66,A -85,B 0,C 180,E1 2869.14,E2 2869.14} C_VEL
LIN {X 0,Y 562.34,Z 580.66,A -85,B 0,C 180,E1 2874.968,E2 2874.968} C_VEL
LIN {X 0,Y 562.366,Z 580.66,A -85,B 0,C 180,E1 2880.004,E2 2880.004} C_VEL
LIN {X 0,Y 562.34,Z 580.66,A -85,B 0,C 180,E1 2885.032,E2 2885.032} C_VEL
LIN {X 0,Y 562.209,Z 580.66,A -85,B 0,C 180,E1 2890.87,E2 2890.87} C_VEL
LIN {X 0,Y 562.163,Z 580.66,A -85,B 0,C 180,E1 2895.628,E2 2895.628} C_VEL
LIN {X 0,Y 562.206,Z 580.66,A -85,B 0,C 180,E1 2900.497,E2 2900.497} C_VEL
LIN {X 0,Y 562.094,Z 580.66,A -85,B 0,C 180,E1 2905.534,E2 2905.534} C_VEL
LIN {X 0,Y 562.07,Z 580.66,A -85,B 0,C 180,E1 2910.789,E2 2910.789} C_VEL
LIN {X 0,Y 562.164,Z 580.66,A -85,B 0,C 180,E1 2916.34,E2 2916.34} C_VEL
LIN {X 0,Y 561.957,Z 580.66,A -85,B 0,C 180,E1 2922.348,E2 2922.348} C_VEL
LIN {X 0,Y 561.962,Z 580.66,A -85,B 0,C 180,E1 2927.661,E2 2927.661} C_VEL
LIN {X 0,Y 562.239,Z 580.66,A -85,B 0,C 180,E1 2933.894,E2 2933.894} C_VEL
LIN {X 0,Y 562.17,Z 580.66,A -85,B 0,C 180,E1 2939.53,E2 2939.53} C_VEL
LIN {X 0,Y 562.069,Z 580.66,A -85,B 0,C 180,E1 2944.472,E2 2944.472} C_VEL
LIN {X 0,Y 562.409,Z 581.204,A -85,B 0,C 180,E1 2949.164,E2 2949.164} C_VEL
LIN {X 0,Y 565.272,Z 597.61,A -85,B 0,C 180,E1 2950.016,E2 2950.016} C_VEL
LIN {X 0,Y 564.576,Z 627.888,A -85,B 0,C 180,E1 2951.863,E2 2951.863} C_VEL
LIN {X 0,Y 563.839,Z 655.285,A -85,B 0,C 180,E1 2954.226,E2 2954.226} C_VEL
LIN {X 0,Y 563.269,Z 678.474,A -85,B 0,C 180,E1 2956.992,E2 2956.992} C_VEL
LIN {X 0,Y 562.933,Z 696.085,A -85,B 0,C 180,E1 2959.933,E2 2959.933} C_VEL
LIN {X 0,Y 562.795,Z 708.94,A -85,B 0,C 180,E1 2963.048,E2 2963.048} C_VEL
LIN {X 0,Y 562.717,Z 716.684,A -85,B 0,C 180,E1 2966.145,E2 2966.145} C_VEL
LIN {X 0,Y 562.655,Z 719.448,A -85,B 0,C 180,E1 2968.459,E2 2968.459} C_VEL
LIN {X 0,Y 562.662,Z 719.385,A -85,B 0,C 180,E1 2971.543,E2 2971.543} C_VEL
LIN {X 0,Y 562.726,Z 714.975,A -85,B 0,C 180,E1 2974.631,E2 2974.631} C_VEL
LIN {X 0,Y 562.835,Z 704.38,A -85,B 0,C 180,E1 2978.12,E2 2978.12} C_VEL
LIN {X 0,Y 563.059,Z 689.181,A -85,B 0,C 180,E1 2981.258,E2 2981.258} C_VEL
LIN {X 0,Y 563.492,Z 668.816,A -85,B 0,C 180,E1 2984.178,E2 2984.178} C_VEL
LIN {X 0,Y 564.139,Z 642.677,A -85,B 0,C 180,E1 2986.87,E2 2986.87} C_VEL
LIN {X 0,Y 564.933,Z 613.037,A -85,B 0,C 180,E1 2989.038,E2 2989.038} C_VEL
LIN {X 0,Y 564.37,Z 588.67,A -85,B 0,C 180,E1 2990.355,E2 2990.355} C_VEL
LIN {X 0,Y 562.404,Z 580.66,A -85,B 0,C 180,E1 2990.834,E2 2990.834} C_VEL
LIN {X 0,Y 562.111,Z 580.66,A -85,B 0,C 180,E1 2997.262,E2 2997.262} C_VEL
LIN {X 0,Y 561.972,Z 580.66,A -85,B 0,C 180,E1 3002.605,E2 3002.605} C_VEL
LIN {X 0,Y 562.121,Z 580.66,A -85,B 0,C 180,E1 3008.28,E2 3008.28} C_VEL
LIN {X 0,Y 561.983,Z 580.66,A -85,B 0,C 180,E1 3014.466,E2 3014.466} C_VEL
LIN {X 0,Y 561.987,Z 580.66,A -85,B 0,C 180,E1 3019.711,E2 3019.711} C_VEL
LIN {X 0,Y 561.974,Z 580.66,A -85,B 0,C 180,E1 3025.539,E2 3025.539} C_VEL
LIN {X 0,Y 562.027,Z 580.66,A -85,B 0,C 180,E1 3030.989,E2 3030.989} C_VEL
LIN {X 0,Y 562.166,Z 580.66,A -85,B 0,C 180,E1 3036.307,E2 3036.307} C_VEL
LIN {X 0,Y 562.318,Z 580.66,A -85,B 0,C 180,E1 3041.145,E2 3041.145} C_VEL
LIN {X 0,Y 561.946,Z 580.66,A -85,B 0,C 180,E1 3045.962,E2 3045.962} C_VEL
LIN {X 0,Y 562.198,Z 580.66,A -85,B 0,C 180,E1 3051.395,E2 3051.395} C_VEL
LIN {X 0,Y 562.349,Z 580.66,A -85,B 0,C 180,E1 3055.363,E2 3055.363} C_VEL
LIN {X 0,Y 562.393,Z 580.66,A -85,B 0,C 180,E1 3059.996,E2 3059.996} C_VEL
LIN {X 0,Y 562.324,Z 580.66,A -85,B 0,C 180,E1 3064.98,E2 3064.98} C_VEL
LIN {X 0,Y 562.357,Z 580.66,A -85,B 0,C 180,E1 3069.292,E2 3069.292} C_VEL
LIN {X 0,Y 562.209,Z 580.66,A -85,B 0,C 180,E1 3074.654,E2 3074.654} C_VEL
LIN {X 0,Y 558.211,Z 580.66,A -85,B 0,C 180,E1 3076.399,E2 3076.399} C_VEL
LIN {X 0,Y 554.286,Z 580.66,A -85,B 0,C 180,E1 3078.168,E2 3078.168} C_VEL
LIN {X 0,Y 554.226,Z 580.66,A -85,B 0,C 180,E1 3084.185,E2 3084.185} C_VEL
LIN {X 0,Y 554.148,Z 580.66,A -85,B 0,C 180,E1 3089.453,E2 3089.453} C_VEL
LIN {X 0,Y 554.084,Z 580.66,A -85,B 0,C 180,E1 3095.012,E2 3095.012} C_VEL
LIN {X 0,Y 554.035,Z 580.66,A -85,B 0,C 180,E1 3100.979,E2 3100.979} C_VEL
LIN {X 0,Y 554.161,Z 580.66,A -85,B 0,C 180,E1 3106.918,E2 3106.918} C_VEL
LIN {X 0,Y 554.118,Z 580.66,A -85,B 0,C 180,E1 3113.049,E2 3113.049} C_VEL
LIN {X 0,Y 554.119,Z 580.66,A -85,B 0,C 180,E1 3118.724,E2 3118.724} C_VEL
LIN {X 0,Y 554.328,Z 581.247,A -85,B 0,C 180,E1 3121.541,E2 3121.541} C_VEL
LIN {X 0,Y 561.1,Z 599.003,A -85,B 0,C 180,E1 3122.167,E2 3122.167} C_VEL
LIN {X 0,Y 560.571,Z 667.716,A -85,B 0,C 180,E1 3123.253,E2 3123.253} C_VEL
LIN {X 0,Y 559.723,Z 704.888,A -85,B 0,C 180,E1 3124.498,E2 3124.498} C_VEL
LIN {X 0,Y 558.616,Z 739.249,A -85,B 0,C 180,E1 3126.284,E2 3126.284} C_VEL
LIN {X 0,Y 557.404,Z 772.137,A -85,B 0,C 180,E1 3128.696,E2 3128.696} C_VEL
LIN {X 0,Y 556.387,Z 800.461,A -85,B 0,C 180,E1 3131.525,E2 3131.525} C_VEL
LIN {X 0,Y 555.62,Z 824.182,A -85,B 0,C 180,E1 3134.674,E2 3134.674} C_VEL
LIN {X 0,Y 555.091,Z 843.715,A -85,B 0,C 180,E1 3138.195,E2 3138.195} C_VEL
LIN {X 0,Y 554.902,Z 857.455,A -85,B 0,C 180,E1 3141.763,E2 3141.763} C_VEL
LIN {X 0,Y 554.754,Z 865.965,A -85,B 0,C 180,E1 3145.302,E2 3145.302} C_VEL
LIN {X 0,Y 554.706,Z 869.508,A -85,B 0,C 180,E1 3148.435,E2 3148.435} C_VEL
LIN {X 0,Y 554.792,Z 869.51,A -85,B 0,C 180,E1 3151.562,E2 3151.562} C_VEL
LIN {X 0,Y 554.777,Z 864.38,A -85,B 0,C 180,E1 3155.519,E2 3155.519} C_VEL
LIN {X 0,Y 554.885,Z 854.841,A -85,B 0,C 180,E1 3159.025,E2 3159.025} C_VEL
LIN {X 0,Y 555.185,Z 838.845,A -85,B 0,C 180,E1 3162.8,E2 3162.8} C_VEL
LIN {X 0,Y 555.714,Z 818.206,A -85,B 0,C 180,E1 3166.214,E2 3166.214} C_VEL
LIN {X 0,Y 556.633,Z 792.346,A -85,B 0,C 180,E1 3169.372,E2 3169.372} C_VEL
LIN {X 0,Y 557.804,Z 762.159,A -85,B 0,C 180,E1 3172.122,E2 3172.122} C_VEL
LIN {X 0,Y 558.986,Z 729.339,A -85,B 0,C 180,E1 3174.3,E2 3174.3} C_VEL
LIN {X 0,Y 560.033,Z 694.818,A -85,B 0,C 180,E1 3175.903,E2 3175.903} C_VEL
LIN {X 0,Y 560.804,Z 659.21,A -85,B 0,C 180,E1 3176.931,E2 3176.931} C_VEL
LIN {X 0,Y 560.508,Z 596.361,A -85,B 0,C 180,E1 3177.902,E2 3177.902} C_VEL
LIN {X 0,Y 554.338,Z 580.66,A -85,B 0,C 180,E1 3178.55,E2 3178.55} C_VEL
LIN {X 0,Y 554.119,Z 580.66,A -85,B 0,C 180,E1 3185.013,E2 3185.013} C_VEL
LIN {X 0,Y 554.026,Z 580.66,A -85,B 0,C 180,E1 3190.983,E2 3190.983} C_VEL
LIN {X 0,Y 554.175,Z 580.66,A -85,B 0,C 180,E1 3196.927,E2 3196.927} C_VEL
LIN {X 0,Y 554.105,Z 580.66,A -85,B 0,C 180,E1 3203.055,E2 3203.055} C_VEL
LIN {X 0,Y 554.105,Z 580.66,A -85,B 0,C 180,E1 3208.73,E2 3208.73} C_VEL
LIN {X 0,Y 554.305,Z 580.66,A -85,B 0,C 180,E1 3214.333,E2 3214.333} C_VEL
LIN {X 0,Y 554.382,Z 580.66,A -85,B 0,C 180,E1 3220.874,E2 3220.874} C_VEL
LIN {X 0,Y 554.106,Z 580.66,A -85,B 0,C 180,E1 3225.769,E2 3225.769} C_VEL
LIN {X 0,Y 554.338,Z 580.66,A -85,B 0,C 180,E1 3230.573,E2 3230.573} C_VEL
LIN {X 0,Y 554.435,Z 580.66,A -85,B 0,C 180,E1 3235.305,E2 3235.305} C_VEL
LIN {X 0,Y 554.465,Z 580.66,A -85,B 0,C 180,E1 3240.004,E2 3240.004} C_VEL
LIN {X 0,Y 554.503,Z 580.66,A -85,B 0,C 180,E1 3244.703,E2 3244.703} C_VEL
LIN {X 0,Y 554.317,Z 580.66,A -85,B 0,C 180,E1 3250.501,E2 3250.501} C_VEL
LIN {X 0,Y 554.254,Z 580.66,A -85,B 0,C 180,E1 3255.857,E2 3255.857} C_VEL
LIN {X 0,Y 554.266,Z 580.66,A -85,B 0,C 180,E1 3260.805,E2 3260.805} C_VEL
LIN {X 0,Y 554.148,Z 580.66,A -85,B 0,C 180,E1 3265.927,E2 3265.927} C_VEL
LIN {X 0,Y 554.137,Z 580.66,A -85,B 0,C 180,E1 3271.279,E2 3271.279} C_VEL
LIN {X 0,Y 554.164,Z 580.66,A -85,B 0,C 180,E1 3276.951,E2 3276.951} C_VEL
LIN {X 0,Y 554.065,Z 580.66,A -85,B 0,C 180,E1 3282.458,E2 3282.458} C_VEL
LIN {X 0,Y 554.1,Z 580.66,A -85,B 0,C 180,E1 3289.024,E2 3289.024} C_VEL
LIN {X 0,Y 554.351,Z 580.66,A -85,B 0,C 180,E1 3295.027,E2 3295.027} C_VEL
LIN {X 0,Y 554.24,Z 580.66,A -85,B 0,C 180,E1 3300.954,E2 3300.954} C_VEL
LIN {X 0,Y 554.207,Z 580.66,A -85,B 0,C 180,E1 3305.811,E2 3305.811} C_VEL
LIN {X 0,Y 554.431,Z 580.925,A -85,B 0,C 180,E1 3308.75,E2 3308.75} C_VEL
LIN {X 0,Y 557.778,Z 598.663,A -85,B 0,C 180,E1 3309.793,E2 3309.793} C_VEL
LIN {X 0,Y 556.935,Z 629.795,A -85,B 0,C 180,E1 3311.747,E2 3311.747} C_VEL
LIN {X 0,Y 556.085,Z 657.2,A -85,B 0,C 180,E1 3314.202,E2 3314.202} C_VEL
LIN {X 0,Y 555.43,Z 679.814,A -85,B 0,C 180,E1 3317.006,E2 3317.006} C_VEL
LIN {X 0,Y 555.064,Z 698.145,A -85,B 0,C 180,E1 3320.209,E2 3320.209} C_VEL
LIN {X 0,Y 554.891,Z 710.152,A -85,B 0,C 180,E1 3323.342,E2 3323.342} C_VEL
LIN {X 0,Y 554.823,Z 717.884,A -85,B 0,C 180,E1 3326.873,E2 3326.873} C_VEL
LIN {X 0,Y 554.8,Z 719.995,A -85,B 0,C 180,E1 3330.001,E2 3330.001} C_VEL
LIN {X 0,Y 554.793,Z 717.744,A -85,B 0,C 180,E1 3333.13,E2 3333.13} C_VEL
LIN {X 0,Y 554.88,Z 709.882,A -85,B 0,C 180,E1 3336.661,E2 3336.661} C_VEL
LIN {X 0,Y 555.095,Z 697.655,A -85,B 0,C 180,E1 3339.8,E2 3339.8} C_VEL
LIN {X 0,Y 555.454,Z 679.196,A -85,B 0,C 180,E1 3342.997,E2 3342.997} C_VEL
LIN {X 0,Y 556.112,Z 656.316,A -85,B 0,C 180,E1 3345.8,E2 3345.8} C_VEL
LIN {X 0,Y 556.941,Z 628.309,A -85,B 0,C 180,E1 3348.272,E2 3348.272} C_VEL
LIN {X 0,Y 557.661,Z 596.636,A -85,B 0,C 180,E1 3350.229,E2 3350.229} C_VEL
LIN {X 0,Y 554.439,Z 580.66,A -85,B 0,C 180,E1 3351.218,E2 3351.218} C_VEL
LIN {X 0,Y 554.179,Z 580.66,A -85,B 0,C 180,E1 3357.676,E2 3357.676} C_VEL
LIN {X 0,Y 554.07,Z 580.66,A -85,B 0,C 180,E1 3363.13,E2 3363.13} C_VEL
LIN {X 0,Y 554.176,Z 580.66,A -85,B 0,C 180,E1 3368.931,E2 3368.931} C_VEL
LIN {X 0,Y 554.127,Z 580.66,A -85,B 0,C 180,E1 3375.268,E2 3375.268} C_VEL
LIN {X 0,Y 554.065,Z 580.66,A -85,B 0,C 180,E1 3381.055,E2 3381.055} C_VEL
LIN {X 0,Y 554.043,Z 580.66,A -85,B 0,C 180,E1 3386.865,E2 3386.865} C_VEL
LIN {X 0,Y 554.161,Z 580.66,A -85,B 0,C 180,E1 3392.32,E2 3392.32} C_VEL
LIN {X 0,Y 554.276,Z 580.66,A -85,B 0,C 180,E1 3398.24,E2 3398.24} C_VEL
LIN {X 0,Y 554.444,Z 580.66,A -85,B 0,C 180,E1 3402.895,E2 3402.895} C_VEL
LIN {X 0,Y 554.326,Z 580.66,A -85,B 0,C 180,E1 3409.51,E2 3409.51} C_VEL
LIN {X 0,Y 554.471,Z 580.66,A -85,B 0,C 180,E1 3415.297,E2 3415.297} C_VEL
LIN {X 0,Y 554.492,Z 580.66,A -85,B 0,C 180,E1 3419.996,E2 3419.996} C_VEL
LIN {X 0,Y 554.49,Z 580.66,A -85,B 0,C 180,E1 3424.694,E2 3424.694} C_VEL
LIN {X 0,Y 554.331,Z 580.66,A -85,B 0,C 180,E1 3430.493,E2 3430.493} C_VEL
LIN {X 0,Y 554.256,Z 580.66,A -85,B 0,C 180,E1 3435.848,E2 3435.848} C_VEL
LIN {X 0,Y 554.286,Z 580.66,A -85,B 0,C 180,E1 3438.168,E2 3438.168} C_VEL
LIN {X 0,Y 553.022,Z 580.66,A -85,B 0,C 180,E1 3439.061,E2 3439.061} C_VEL
LIN {X 0,Y 546.403,Z 580.66,A -85,B 0,C 180,E1 3441.49,E2 3441.49} C_VEL
LIN {X 0,Y 546.296,Z 580.66,A -85,B 0,C 180,E1 3441.721,E2 3441.721} C_VEL
LIN {X 0,Y 546.283,Z 580.66,A -85,B 0,C 180,E1 3447.513,E2 3447.513} C_VEL
LIN {X 0,Y 546.181,Z 580.66,A -85,B 0,C 180,E1 3453.734,E2 3453.734} C_VEL
LIN {X 0,Y 546.127,Z 580.66,A -85,B 0,C 180,E1 3459.609,E2 3459.609} C_VEL
LIN {X 0,Y 546.197,Z 580.66,A -85,B 0,C 180,E1 3466.131,E2 3466.131} C_VEL
LIN {X 0,Y 546.217,Z 580.66,A -85,B 0,C 180,E1 3472.423,E2 3472.423} C_VEL
LIN {X 0,Y 546.182,Z 580.66,A -85,B 0,C 180,E1 3478.217,E2 3478.217} C_VEL
LIN {X 0,Y 546.401,Z 580.66,A -85,B 0,C 180,E1 3481.073,E2 3481.073} C_VEL
LIN {X 0,Y 554.162,Z 602.241,A -85,B 0,C 180,E1 3481.834,E2 3481.834} C_VEL
LIN {X 0,Y 553.539,Z 666.971,A -85,B 0,C 180,E1 3482.865,E2 3482.865} C_VEL
LIN {X 0,Y 552.554,Z 703.094,A -85,B 0,C 180,E1 3484.063,E2 3484.063} C_VEL
LIN {X 0,Y 551.288,Z 738.676,A -85,B 0,C 180,E1 3485.913,E2 3485.913} C_VEL
LIN {X 0,Y 549.919,Z 772.135,A -85,B 0,C 180,E1 3488.392,E2 3488.392} C_VEL
LIN {X 0,Y 548.727,Z 800.737,A -85,B 0,C 180,E1 3491.29,E2 3491.29} C_VEL
LIN {X 0,Y 547.82,Z 824.816,A -85,B 0,C 180,E1 3494.549,E2 3494.549} C_VEL
LIN {X 0,Y 547.24,Z 843.715,A -85,B 0,C 180,E1 3498.023,E2 3498.023} C_VEL
LIN {X 0,Y 547.039,Z 857.455,A -85,B 0,C 180,E1 3501.644,E2 3501.644} C_VEL
LIN {X 0,Y 546.86,Z 866.038,A -85,B 0,C 180,E1 3505.283,E2 3505.283} C_VEL
LIN {X 0,Y 546.805,Z 869.508,A -85,B 0,C 180,E1 3508.412,E2 3508.412} C_VEL
LIN {X 0,Y 546.888,Z 869.51,A -85,B 0,C 180,E1 3511.585,E2 3511.585} C_VEL
LIN {X 0,Y 546.901,Z 864.614,A -85,B 0,C 180,E1 3515.479,E2 3515.479} C_VEL
LIN {X 0,Y 547.017,Z 854.841,A -85,B 0,C 180,E1 3519.156,E2 3519.156} C_VEL
LIN {X 0,Y 547.338,Z 839.827,A -85,B 0,C 180,E1 3522.783,E2 3522.783} C_VEL
LIN {X 0,Y 547.933,Z 819.649,A -85,B 0,C 180,E1 3526.245,E2 3526.245} C_VEL
LIN {X 0,Y 548.963,Z 794.048,A -85,B 0,C 180,E1 3529.468,E2 3529.468} C_VEL
LIN {X 0,Y 550.214,Z 764.695,A -85,B 0,C 180,E1 3532.23,E2 3532.23} C_VEL
LIN {X 0,Y 551.638,Z 730.847,A -85,B 0,C 180,E1 3534.559,E2 3534.559} C_VEL
LIN {X 0,Y 552.846,Z 696.06,A -85,B 0,C 180,E1 3536.216,E2 3536.216} C_VEL
LIN {X 0,Y 553.733,Z 660.665,A -85,B 0,C 180,E1 3537.271,E2 3537.271} C_VEL
LIN {X 0,Y 553.493,Z 598.444,A -85,B 0,C 180,E1 3538.258,E2 3538.258} C_VEL
LIN {X 0,Y 546.364,Z 580.66,A -85,B 0,C 180,E1 3539.007,E2 3539.007} C_VEL
LIN {X 0,Y 546.201,Z 580.66,A -85,B 0,C 180,E1 3543.747,E2 3543.747} C_VEL
LIN {X 0,Y 546.122,Z 580.66,A -85,B 0,C 180,E1 3549.613,E2 3549.613} C_VEL
LIN {X 0,Y 546.234,Z 580.66,A -85,B 0,C 180,E1 3556.143,E2 3556.143} C_VEL
LIN {X 0,Y 546.205,Z 580.66,A -85,B 0,C 180,E1 3562.429,E2 3562.429} C_VEL
LIN {X 0,Y 546.171,Z 580.66,A -85,B 0,C 180,E1 3568.223,E2 3568.223} C_VEL
LIN {X 0,Y 546.296,Z 580.66,A -85,B 0,C 180,E1 3573.682,E2 3573.682} C_VEL
LIN {X 0,Y 546.39,Z 580.66,A -85,B 0,C 180,E1 3578.891,E2 3578.891} C_VEL
LIN {X 0,Y 546.396,Z 580.66,A -85,B 0,C 180,E1 3583.918,E2 3583.918} C_VEL
LIN {X 0,Y 546.437,Z 580.66,A -85,B 0,C 180,E1 3590.435,E2 3590.435} C_VEL
LIN {X 0,Y 546.508,Z 580.66,A -85,B 0,C 180,E1 3595.789,E2 3595.789} C_VEL
LIN {X 0,Y 546.565,Z 580.66,A -85,B 0,C 180,E1 3600.004,E2 3600.004} C_VEL
LIN {X 0,Y 546.59,Z 580.66,A -85,B 0,C 180,E1 3604.771,E2 3604.771} C_VEL
LIN {X 0,Y 546.493,Z 580.66,A -85,B 0,C 180,E1 3609.573,E2 3609.573} C_VEL
LIN {X 0,Y 546.454,Z 580.66,A -85,B 0,C 180,E1 3614.444,E2 3614.444} C_VEL
LIN {X 0,Y 546.402,Z 580.66,A -85,B 0,C 180,E1 3619.597,E2 3619.597} C_VEL
LIN {X 0,Y 546.296,Z 580.66,A -85,B 0,C 180,E1 3624.569,E2 3624.569} C_VEL
LIN {X 0,Y 546.193,Z 580.66,A -85,B 0,C 180,E1 3630.764,E2 3630.764} C_VEL
LIN {X 0,Y 546.238,Z 580.66,A -85,B 0,C 180,E1 3636.508,E2 3636.508} C_VEL
LIN {X 0,Y 546.15,Z 580.66,A -85,B 0,C 180,E1 3641.713,E2 3641.713} C_VEL
LIN {X 0,Y 546.162,Z 580.66,A -85,B 0,C 180,E1 3648.465,E2 3648.465} C_VEL
LIN {X 0,Y 546.325,Z 580.66,A -85,B 0,C 180,E1 3654.413,E2 3654.413} C_VEL
LIN {X 0,Y 546.265,Z 580.66,A -85,B 0,C 180,E1 3660.075,E2 3660.075} C_VEL
LIN {X 0,Y 546.307,Z 580.66,A -85,B 0,C 180,E1 3666.154,E2 3666.154} C_VEL
LIN {X 0,Y 546.502,Z 581.337,A -85,B 0,C 180,E1 3668.319,E2 3668.319} C_VEL
LIN {X 0,Y 550.612,Z 600.619,A -85,B 0,C 180,E1 3669.51,E2 3669.51} C_VEL
LIN {X 0,Y 549.439,Z 629.852,A -85,B 0,C 180,E1 3671.449,E2 3671.449} C_VEL
LIN {X 0,Y 548.335,Z 659.048,A -85,B 0,C 180,E1 3674.172,E2 3674.172} C_VEL
LIN {X 0,Y 547.602,Z 681.136,A -85,B 0,C 180,E1 3677.02,E2 3677.02} C_VEL
LIN {X 0,Y 547.211,Z 698.36,A -85,B 0,C 180,E1 3680.112,E2 3680.112} C_VEL
LIN {X 0,Y 547.011,Z 711.298,A -85,B 0,C 180,E1 3683.645,E2 3683.645} C_VEL
LIN {X 0,Y 546.923,Z 717.884,A -85,B 0,C 180,E1 3686.828,E2 3686.828} C_VEL
LIN {X 0,Y 546.9,Z 719.995,A -85,B 0,C 180,E1 3690.001,E2 3690.001} C_VEL
LIN {X 0,Y 546.995,Z 716.569,A -85,B 0,C 180,E1 3693.946,E2 3693.946} C_VEL
LIN {X 0,Y 547.077,Z 707.289,A -85,B 0,C 180,E1 3697.555,E2 3697.555} C_VEL
LIN {X 0,Y 547.323,Z 692.777,A -85,B 0,C 180,E1 3700.921,E2 3700.921} C_VEL
LIN {X 0,Y 547.865,Z 673.429,A -85,B 0,C 180,E1 3703.995,E2 3703.995} C_VEL
LIN {X 0,Y 548.674,Z 648.225,A -85,B 0,C 180,E1 3706.844,E2 3706.844} C_VEL
LIN {X 0,Y 549.947,Z 618.565,A -85,B 0,C 180,E1 3709.292,E2 3709.292} C_VEL
LIN {X 0,Y 550.067,Z 593.691,A -85,B 0,C 180,E1 3710.802,E2 3710.802} C_VEL
LIN {X 0,Y 546.472,Z 580.66,A -85,B 0,C 180,E1 3711.679,E2 3711.679} C_VEL
LIN {X 0,Y 546.262,Z 580.66,A -85,B 0,C 180,E1 3717.502,E2 3717.502} C_VEL
LIN {X 0,Y 546.13,Z 580.66,A -85,B 0,C 180,E1 3723.72,E2 3723.72} C_VEL
LIN {X 0,Y 546.217,Z 580.66,A -85,B 0,C 180,E1 3729.609,E2 3729.609} C_VEL
LIN {X 0,Y 546.188,Z 580.66,A -85,B 0,C 180,E1 3736.126,E2 3736.126} C_VEL
LIN {X 0,Y 546.169,Z 580.66,A -85,B 0,C 180,E1 3742.415,E2 3742.415} C_VEL
LIN {X 0,Y 546.14,Z 580.66,A -85,B 0,C 180,E1 3748.21,E2 3748.21} C_VEL
LIN {X 0,Y 546.266,Z 580.66,A -85,B 0,C 180,E1 3753.671,E2 3753.671} C_VEL
LIN {X 0,Y 546.427,Z 580.66,A -85,B 0,C 180,E1 3758.883,E2 3758.883} C_VEL
LIN {X 0,Y 546.363,Z 580.66,A -85,B 0,C 180,E1 3763.908,E2 3763.908} C_VEL
LIN {X 0,Y 546.428,Z 580.66,A -85,B 0,C 180,E1 3770.426,E2 3770.426} C_VEL
LIN {X 0,Y 546.531,Z 580.66,A -85,B 0,C 180,E1 3775.796,E2 3775.796} C_VEL
LIN {X 0,Y 546.592,Z 580.66,A -85,B 0,C 180,E1 3779.996,E2 3779.996} C_VEL
LIN {X 0,Y 546.592,Z 580.66,A -85,B 0,C 180,E1 3784.762,E2 3784.762} C_VEL
LIN {X 0,Y 546.51,Z 580.66,A -85,B 0,C 180,E1 3789.564,E2 3789.564} C_VEL
LIN {X 0,Y 546.461,Z 580.66,A -85,B 0,C 180,E1 3794.435,E2 3794.435} C_VEL
LIN {X 0,Y 546.397,Z 580.66,A -85,B 0,C 180,E1 3799.587,E2 3799.587} C_VEL
LIN {X 0,Y 546.296,Z 580.66,A -85,B 0,C 180,E1 3801.721,E2 3801.721} C_VEL
LIN {X 0,Y 542.298,Z 580.66,A -85,B 0,C 180,E1 3803.508,E2 3803.508} C_VEL
LIN {X 0,Y 538.313,Z 580.66,A -85,B 0,C 180,E1 3805.321,E2 3805.321} C_VEL
LIN {X 0,Y 538.258,Z 580.66,A -85,B 0,C 180,E1 3810.413,E2 3810.413} C_VEL
LIN {X 0,Y 538.17,Z 580.66,A -85,B 0,C 180,E1 3816.208,E2 3816.208} C_VEL
LIN {X 0,Y 538.142,Z 580.66,A -85,B 0,C 180,E1 3822.465,E2 3822.465} C_VEL
LIN {X 0,Y 538.223,Z 580.66,A -85,B 0,C 180,E1 3827.535,E2 3827.535} C_VEL
LIN {X 0,Y 538.248,Z 580.66,A -85,B 0,C 180,E1 3833.791,E2 3833.791} C_VEL
LIN {X 0,Y 538.369,Z 580.66,A -85,B 0,C 180,E1 3840.433,E2 3840.433} C_VEL
LIN {X 0,Y 538.412,Z 580.66,A -85,B 0,C 180,E1 3840.61,E2 3840.61} C_VEL
LIN {X 0,Y 547.03,Z 602.382,A -85,B 0,C 180,E1 3841.436,E2 3841.436} C_VEL
LIN {X 0,Y 546.534,Z 666.807,A -85,B 0,C 180,E1 3842.483,E2 3842.483} C_VEL
LIN {X 0,Y 545.363,Z 703.952,A -85,B 0,C 180,E1 3843.734,E2 3843.734} C_VEL
LIN {X 0,Y 543.974,Z 738.266,A -85,B 0,C 180,E1 3845.542,E2 3845.542} C_VEL
LIN {X 0,Y 542.473,Z 770.946,A -85,B 0,C 180,E1 3847.972,E2 3847.972} C_VEL
LIN {X 0,Y 541.185,Z 798.983,A -85,B 0,C 180,E1 3850.807,E2 3850.807} C_VEL
LIN {X 0,Y 540.097,Z 823.635,A -85,B 0,C 180,E1 3854.137,E2 3854.137} C_VEL
LIN {X 0,Y 539.423,Z 843.714,A -85,B 0,C 180,E1 3857.847,E2 3857.847} C_VEL
LIN {X 0,Y 539.154,Z 857.455,A -85,B 0,C 180,E1 3861.521,E2 3861.521} C_VEL
LIN {X 0,Y 538.968,Z 865.963,A -85,B 0,C 180,E1 3865.164,E2 3865.164} C_VEL
LIN {X 0,Y 538.919,Z 869.508,A -85,B 0,C 180,E1 3868.389,E2 3868.389} C_VEL
LIN {X 0,Y 538.997,Z 869.511,A -85,B 0,C 180,E1 3871.608,E2 3871.608} C_VEL
LIN {X 0,Y 539.051,Z 865.969,A -85,B 0,C 180,E1 3874.832,E2 3874.832} C_VEL
LIN {X 0,Y 539.147,Z 856.179,A -85,B 0,C 180,E1 3878.883,E2 3878.883} C_VEL
LIN {X 0,Y 539.455,Z 841.784,A -85,B 0,C 180,E1 3882.561,E2 3882.561} C_VEL
LIN {X 0,Y 540.105,Z 822.327,A -85,B 0,C 180,E1 3886.069,E2 3886.069} C_VEL
LIN {X 0,Y 541.212,Z 797.249,A -85,B 0,C 180,E1 3889.401,E2 3889.401} C_VEL
LIN {X 0,Y 542.611,Z 767.22,A -85,B 0,C 180,E1 3892.343,E2 3892.343} C_VEL
LIN {X 0,Y 544.19,Z 734.908,A -85,B 0,C 180,E1 3894.664,E2 3894.664} C_VEL
LIN {X 0,Y 545.654,Z 698.895,A -85,B 0,C 180,E1 3896.476,E2 3896.476} C_VEL
LIN {X 0,Y 546.653,Z 663.057,A -85,B 0,C 180,E1 3897.6,E2 3897.6} C_VEL
LIN {X 0,Y 546.662,Z 600.83,A -85,B 0,C 180,E1 3898.608,E2 3898.608} C_VEL
LIN {X 0,Y 538.382,Z 580.66,A -85,B 0,C 180,E1 3899.425,E2 3899.425} C_VEL
LIN {X 0,Y 538.196,Z 580.66,A -85,B 0,C 180,E1 3905.34,E2 3905.34} C_VEL
LIN {X 0,Y 538.131,Z 580.66,A -85,B 0,C 180,E1 3910.574,E2 3910.574} C_VEL
LIN {X 0,Y 538.261,Z 580.66,A -85,B 0,C 180,E1 3916.996,E2 3916.996} C_VEL
LIN {X 0,Y 538.287,Z 580.66,A -85,B 0,C 180,E1 3921.954,E2 3921.954} C_VEL
LIN {X 0,Y 538.198,Z 580.66,A -85,B 0,C 180,E1 3927.696,E2 3927.696} C_VEL
LIN {X 0,Y 538.375,Z 580.66,A -85,B 0,C 180,E1 3933.264,E2 3933.264} C_VEL
LIN {X 0,Y 538.432,Z 580.66,A -85,B 0,C 180,E1 3938.563,E2 3938.563} C_VEL
LIN {X 0,Y 538.485,Z 580.66,A -85,B 0,C 180,E1 3943.675,E2 3943.675} C_VEL
LIN {X 0,Y 538.52,Z 580.66,A -85,B 0,C 180,E1 3950.293,E2 3950.293} C_VEL
LIN {X 0,Y 538.654,Z 580.66,A -85,B 0,C 180,E1 3955.167,E2 3955.167} C_VEL
LIN {X 0,Y 538.683,Z 580.66,A -85,B 0,C 180,E1 3960.004,E2 3960.004} C_VEL
LIN {X 0,Y 538.676,Z 580.66,A -85,B 0,C 180,E1 3964.841,E2 3964.841} C_VEL
LIN {X 0,Y 538.514,Z 580.66,A -85,B 0,C 180,E1 3970.266,E2 3970.266} C_VEL
LIN {X 0,Y 538.519,Z 580.66,A -85,B 0,C 180,E1 3974.662,E2 3974.662} C_VEL
LIN {X 0,Y 538.496,Z 580.66,A -85,B 0,C 180,E1 3979.723,E2 3979.723} C_VEL
LIN {X 0,Y 538.298,Z 580.66,A -85,B 0,C 180,E1 3985.841,E2 3985.841} C_VEL
LIN {X 0,Y 538.3,Z 580.66,A -85,B 0,C 180,E1 3990.421,E2 3990.421} C_VEL
LIN {X 0,Y 538.338,Z 580.66,A -85,B 0,C 180,E1 3996.206,E2 3996.206} C_VEL
LIN {X 0,Y 538.117,Z 580.66,A -85,B 0,C 180,E1 4002.48,E2 4002.48} C_VEL
LIN {X 0,Y 538.121,Z 580.66,A -85,B 0,C 180,E1 4007.529,E2 4007.529} C_VEL
LIN {X 0,Y 538.379,Z 580.66,A -85,B 0,C 180,E1 4013.805,E2 4013.805} C_VEL
LIN {X 0,Y 538.36,Z 580.66,A -85,B 0,C 180,E1 4019.59,E2 4019.59} C_VEL
LIN {X 0,Y 538.323,Z 580.66,A -85,B 0,C 180,E1 4025.049,E2 4025.049} C_VEL
LIN {X 0,Y 538.54,Z 580.988,A -85,B 0,C 180,E1 4027.833,E2 4027.833} C_VEL
LIN {X 0,Y 543.53,Z 600.77,A -85,B 0,C 180,E1 4029.11,E2 4029.11} C_VEL
LIN {X 0,Y 542.286,Z 630.068,A -85,B 0,C 180,E1 4031.063,E2 4031.063} C_VEL
LIN {X 0,Y 540.904,Z 656.272,A -85,B 0,C 180,E1 4033.538,E2 4033.538} C_VEL
LIN {X 0,Y 539.808,Z 681.131,A -85,B 0,C 180,E1 4036.829,E2 4036.829} C_VEL
LIN {X 0,Y 539.338,Z 698.715,A -85,B 0,C 180,E1 4040.047,E2 4040.047} C_VEL
LIN {X 0,Y 539.114,Z 711.296,A -85,B 0,C 180,E1 4043.552,E2 4043.552} C_VEL
LIN {X 0,Y 539.038,Z 717.884,A -85,B 0,C 180,E1 4046.781,E2 4046.781} C_VEL
LIN {X 0,Y 539.007,Z 719.995,A -85,B 0,C 180,E1 4050.001,E2 4050.001} C_VEL
LIN {X 0,Y 539.075,Z 716.825,A -85,B 0,C 180,E1 4053.836,E2 4053.836} C_VEL
LIN {X 0,Y 539.181,Z 708.627,A -85,B 0,C 180,E1 4057.261,E2 4057.261} C_VEL
LIN {X 0,Y 539.459,Z 694.391,A -85,B 0,C 180,E1 4060.773,E2 4060.773} C_VEL
LIN {X 0,Y 540.047,Z 674.911,A -85,B 0,C 180,E1 4063.994,E2 4063.994} C_VEL
LIN {X 0,Y 541.179,Z 651.607,A -85,B 0,C 180,E1 4066.875,E2 4066.875} C_VEL
LIN {X 0,Y 542.538,Z 624.914,A -85,B 0,C 180,E1 4069.248,E2 4069.248} C_VEL
LIN {X 0,Y 542.832,Z 595.289,A -85,B 0,C 180,E1 4071.137,E2 4071.137} C_VEL
LIN {X 0,Y 538.483,Z 580.66,A -85,B 0,C 180,E1 4072.164,E2 4072.164} C_VEL
LIN {X 0,Y 538.372,Z 580.66,A -85,B 0,C 180,E1 4076.742,E2 4076.742} C_VEL
LIN {X 0,Y 538.208,Z 580.66,A -85,B 0,C 180,E1 4082.435,E2 4082.435} C_VEL
LIN {X 0,Y 538.344,Z 580.66,A -85,B 0,C 180,E1 4088.225,E2 4088.225} C_VEL
LIN {X 0,Y 538.161,Z 580.66,A -85,B 0,C 180,E1 4094.697,E2 4094.697} C_VEL
LIN {X 0,Y 538.193,Z 580.66,A -85,B 0,C 180,E1 4099.676,E2 4099.676} C_VEL
LIN {X 0,Y 538.159,Z 580.66,A -85,B 0,C 180,E1 4105.754,E2 4105.754} C_VEL
LIN {X 0,Y 538.259,Z 580.66,A -85,B 0,C 180,E1 4111.428,E2 4111.428} C_VEL
LIN {X 0,Y 538.402,Z 580.66,A -85,B 0,C 180,E1 4116.811,E2 4116.811} C_VEL
LIN {X 0,Y 538.567,Z 580.66,A -85,B 0,C 180,E1 4121.982,E2 4121.982} C_VEL
LIN {X 0,Y 538.458,Z 580.66,A -85,B 0,C 180,E1 4128.644,E2 4128.644} C_VEL
LIN {X 0,Y 538.775,Z 580.66,A -85,B 0,C 180,E1 4133.541,E2 4133.541} C_VEL
LIN {X 0,Y 538.887,Z 580.66,A -85,B 0,C 180,E1 4138.386,E2 4138.386} C_VEL
LIN {X 0,Y 538.678,Z 580.66,A -85,B 0,C 180,E1 4144.832,E2 4144.832} C_VEL
LIN {X 0,Y 538.517,Z 580.66,A -85,B 0,C 180,E1 4150.251,E2 4150.251} C_VEL
LIN {X 0,Y 538.526,Z 580.66,A -85,B 0,C 180,E1 4154.652,E2 4154.652} C_VEL
LIN {X 0,Y 538.492,Z 580.66,A -85,B 0,C 180,E1 4159.713,E2 4159.713} C_VEL
LIN {X 0,Y 538.313,Z 580.66,A -85,B 0,C 180,E1 4165.321,E2 4165.321} C_VEL
LIN {X 0,Y 537.014,Z 580.66,A -85,B 0,C 180,E1 4166.244,E2 4166.244} C_VEL
LIN {X 0,Y 530.424,Z 580.66,A -85,B 0,C 180,E1 4168.756,E2 4168.756} C_VEL
LIN {X 0,Y 530.355,Z 580.66,A -85,B 0,C 180,E1 4168.994,E2 4168.994} C_VEL
LIN {X 0,Y 530.288,Z 580.66,A -85,B 0,C 180,E1 4174.816,E2 4174.816} C_VEL
LIN {X 0,Y 530.198,Z 580.66,A -85,B 0,C 180,E1 4181.049,E2 4181.049} C_VEL
LIN {X 0,Y 530.331,Z 580.66,A -85,B 0,C 180,E1 4186.749,E2 4186.749} C_VEL
LIN {X 0,Y 530.302,Z 580.66,A -85,B 0,C 180,E1 4193.066,E2 4193.066} C_VEL
LIN {X 0,Y 530.437,Z 580.66,A -85,B 0,C 180,E1 4199.673,E2 4199.673} C_VEL
LIN {X 0,Y 530.482,Z 581.201,A -85,B 0,C 180,E1 4200.181,E2 4200.181} C_VEL
LIN {X 0,Y 540.23,Z 606.9,A -85,B 0,C 180,E1 4201.109,E2 4201.109} C_VEL
LIN {X 0,Y 539.445,Z 668.199,A -85,B 0,C 180,E1 4202.13,E2 4202.13} C_VEL
LIN {X 0,Y 538.201,Z 705.284,A -85,B 0,C 180,E1 4203.419,E2 4203.419} C_VEL
LIN {X 0,Y 536.616,Z 739.963,A -85,B 0,C 180,E1 4205.295,E2 4205.295} C_VEL
LIN {X 0,Y 534.882,Z 773.48,A -85,B 0,C 180,E1 4207.88,E2 4207.88} C_VEL
LIN {X 0,Y 533.465,Z 800.736,A -85,B 0,C 180,E1 4210.734,E2 4210.734} C_VEL
LIN {X 0,Y 532.286,Z 824.96,A -85,B 0,C 180,E1 4214.11,E2 4214.11} C_VEL
LIN {X 0,Y 531.592,Z 843.714,A -85,B 0,C 180,E1 4217.665,E2 4217.665} C_VEL
LIN {X 0,Y 531.27,Z 857.455,A -85,B 0,C 180,E1 4221.394,E2 4221.394} C_VEL
LIN {X 0,Y 531.097,Z 865.963,A -85,B 0,C 180,E1 4225.092,E2 4225.092} C_VEL
LIN {X 0,Y 531.018,Z 869.509,A -85,B 0,C 180,E1 4228.365,E2 4228.365} C_VEL
LIN {X 0,Y 531.093,Z 869.511,A -85,B 0,C 180,E1 4231.632,E2 4231.632} C_VEL
LIN {X 0,Y 531.171,Z 865.968,A -85,B 0,C 180,E1 4234.904,E2 4234.904} C_VEL
LIN {X 0,Y 531.283,Z 856.178,A -85,B 0,C 180,E1 4239.016,E2 4239.016} C_VEL
LIN {X 0,Y 531.625,Z 841.783,A -85,B 0,C 180,E1 4242.749,E2 4242.749} C_VEL
LIN {X 0,Y 532.371,Z 822.326,A -85,B 0,C 180,E1 4246.309,E2 4246.309} C_VEL
LIN {X 0,Y 533.616,Z 797.249,A -85,B 0,C 180,E1 4249.688,E2 4249.688} C_VEL
LIN {X 0,Y 535.174,Z 767.771,A -85,B 0,C 180,E1 4252.622,E2 4252.622} C_VEL
LIN {X 0,Y 536.917,Z 734.905,A -85,B 0,C 180,E1 4255.021,E2 4255.021} C_VEL
LIN {X 0,Y 538.516,Z 700.247,A -85,B 0,C 180,E1 4256.798,E2 4256.798} C_VEL
LIN {X 0,Y 539.666,Z 663.057,A -85,B 0,C 180,E1 4257.988,E2 4257.988} C_VEL
LIN {X 0,Y 539.459,Z 602.567,A -85,B 0,C 180,E1 4259,E2 4259} C_VEL
LIN {X 0,Y 530.445,Z 580.66,A -85,B 0,C 180,E1 4259.882,E2 4259.882} C_VEL
LIN {X 0,Y 530.307,Z 580.66,A -85,B 0,C 180,E1 4264.818,E2 4264.818} C_VEL
LIN {X 0,Y 530.185,Z 580.66,A -85,B 0,C 180,E1 4271.054,E2 4271.054} C_VEL
LIN {X 0,Y 530.354,Z 580.66,A -85,B 0,C 180,E1 4276.76,E2 4276.76} C_VEL
LIN {X 0,Y 530.292,Z 580.66,A -85,B 0,C 180,E1 4283.167,E2 4283.167} C_VEL
LIN {X 0,Y 530.299,Z 580.66,A -85,B 0,C 180,E1 4289.081,E2 4289.081} C_VEL
LIN {X 0,Y 530.483,Z 580.66,A -85,B 0,C 180,E1 4294.657,E2 4294.657} C_VEL
LIN {X 0,Y 530.637,Z 580.66,A -85,B 0,C 180,E1 4300.311,E2 4300.311} C_VEL
LIN {X 0,Y 530.352,Z 580.66,A -85,B 0,C 180,E1 4306.069,E2 4306.069} C_VEL
LIN {X 0,Y 530.611,Z 580.66,A -85,B 0,C 180,E1 4311.802,E2 4311.802} C_VEL
LIN {X 0,Y 530.721,Z 580.66,A -85,B 0,C 180,E1 4316.798,E2 4316.798} C_VEL
LIN {X 0,Y 530.738,Z 580.66,A -85,B 0,C 180,E1 4321.639,E2 4321.639} C_VEL
LIN {X 0,Y 530.674,Z 580.66,A -85,B 0,C 180,E1 4326.558,E2 4326.558} C_VEL
LIN {X 0,Y 530.588,Z 580.66,A -85,B 0,C 180,E1 4331.527,E2 4331.527} C_VEL
LIN {X 0,Y 530.559,Z 580.66,A -85,B 0,C 180,E1 4336.585,E2 4336.585} C_VEL
LIN {X 0,Y 530.52,Z 580.66,A -85,B 0,C 180,E1 4341.782,E2 4341.782} C_VEL
LIN {X 0,Y 530.336,Z 580.66,A -85,B 0,C 180,E1 4347.752,E2 4347.752} C_VEL
LIN {X 0,Y 530.446,Z 580.66,A -85,B 0,C 180,E1 4354.137,E2 4354.137} C_VEL
LIN {X 0,Y 530.299,Z 580.66,A -85,B 0,C 180,E1 4359.571,E2 4359.571} C_VEL
LIN {X 0,Y 530.123,Z 580.66,A -85,B 0,C 180,E1 4365.568,E2 4365.568} C_VEL
LIN {X 0,Y 530.318,Z 580.66,A -85,B 0,C 180,E1 4371.093,E2 4371.093} C_VEL
LIN {X 0,Y 530.445,Z 580.66,A -85,B 0,C 180,E1 4377.161,E2 4377.161} C_VEL
LIN {X 0,Y 530.325,Z 580.66,A -85,B 0,C 180,E1 4382.822,E2 4382.822} C_VEL
LIN {X 0,Y 530.565,Z 581.059,A -85,B 0,C 180,E1 4387.345,E2 4387.345} C_VEL
LIN {X 0,Y 536.463,Z 602.201,A -85,B 0,C 180,E1 4388.768,E2 4388.768} C_VEL
LIN {X 0,Y 535.032,Z 631.999,A -85,B 0,C 180,E1 4390.796,E2 4390.796} C_VEL
LIN {X 0,Y 533.515,Z 657.971,A -85,B 0,C 180,E1 4393.312,E2 4393.312} C_VEL
LIN {X 0,Y 532.241,Z 680.968,A -85,B 0,C 180,E1 4396.429,E2 4396.429} C_VEL
LIN {X 0,Y 531.481,Z 698.044,A -85,B 0,C 180,E1 4399.725,E2 4399.725} C_VEL
LIN {X 0,Y 531.235,Z 711.294,A -85,B 0,C 180,E1 4403.456,E2 4403.456} C_VEL
LIN {X 0,Y 531.137,Z 717.884,A -85,B 0,C 180,E1 4406.733,E2 4406.733} C_VEL
LIN {X 0,Y 531.107,Z 719.995,A -85,B 0,C 180,E1 4410.002,E2 4410.002} C_VEL
LIN {X 0,Y 531.171,Z 716.839,A -85,B 0,C 180,E1 4413.883,E2 4413.883} C_VEL
LIN {X 0,Y 531.304,Z 708.63,A -85,B 0,C 180,E1 4417.369,E2 4417.369} C_VEL
LIN {X 0,Y 531.686,Z 693.789,A -85,B 0,C 180,E1 4421.125,E2 4421.125} C_VEL
LIN {X 0,Y 532.594,Z 674.636,A -85,B 0,C 180,E1 4424.456,E2 4424.456} C_VEL
LIN {X 0,Y 533.852,Z 651.543,A -85,B 0,C 180,E1 4427.302,E2 4427.302} C_VEL
LIN {X 0,Y 535.452,Z 624.095,A -85,B 0,C 180,E1 4429.729,E2 4429.729} C_VEL
LIN {X 0,Y 536.002,Z 598.543,A -85,B 0,C 180,E1 4431.374,E2 4431.374} C_VEL
LIN {X 0,Y 530.55,Z 580.66,A -85,B 0,C 180,E1 4432.643,E2 4432.643} C_VEL
LIN {X 0,Y 530.358,Z 580.66,A -85,B 0,C 180,E1 4437.743,E2 4437.743} C_VEL
LIN {X 0,Y 530.302,Z 580.66,A -85,B 0,C 180,E1 4444.102,E2 4444.102} C_VEL
LIN {X 0,Y 530.292,Z 580.66,A -85,B 0,C 180,E1 4449.561,E2 4449.561} C_VEL
LIN {X 0,Y 530.286,Z 580.66,A -85,B 0,C 180,E1 4455.545,E2 4455.545} C_VEL
LIN {X 0,Y 530.244,Z 580.66,A -85,B 0,C 180,E1 4461.079,E2 4461.079} C_VEL
LIN {X 0,Y 530.241,Z 580.66,A -85,B 0,C 180,E1 4467.139,E2 4467.139} C_VEL
LIN {X 0,Y 530.382,Z 580.66,A -85,B 0,C 180,E1 4472.818,E2 4472.818} C_VEL
LIN {X 0,Y 530.552,Z 580.66,A -85,B 0,C 180,E1 4478.219,E2 4478.219} C_VEL
LIN {X 0,Y 530.564,Z 580.66,A -85,B 0,C 180,E1 4483.415,E2 4483.415} C_VEL
LIN {X 0,Y 530.588,Z 580.66,A -85,B 0,C 180,E1 4490.137,E2 4490.137} C_VEL
LIN {X 0,Y 530.785,Z 580.66,A -85,B 0,C 180,E1 4495.086,E2 4495.086} C_VEL
LIN {X 0,Y 530.809,Z 580.66,A -85,B 0,C 180,E1 4499.995,E2 4499.995} C_VEL
LIN {X 0,Y 530.763,Z 580.66,A -85,B 0,C 180,E1 4504.905,E2 4504.905} C_VEL
LIN {X 0,Y 530.679,Z 580.66,A -85,B 0,C 180,E1 4509.852,E2 4509.852} C_VEL
LIN {X 0,Y 530.608,Z 580.66,A -85,B 0,C 180,E1 4514.876,E2 4514.876} C_VEL
LIN {X 0,Y 530.544,Z 580.66,A -85,B 0,C 180,E1 4520.021,E2 4520.021} C_VEL
LIN {X 0,Y 530.437,Z 580.66,A -85,B 0,C 180,E1 4525.345,E2 4525.345} C_VEL
LIN {X 0,Y 530.355,Z 580.66,A -85,B 0,C 180,E1 4528.994,E2 4528.994} C_VEL
LIN {X 0,Y 527.841,Z 580.66,A -85,B 0,C 180,E1 4530.389,E2 4530.389} C_VEL
LIN {X 0,Y 522.454,Z 580.66,A -85,B 0,C 180,E1 4532.479,E2 4532.479} C_VEL
LIN {X 0,Y 522.386,Z 580.66,A -85,B 0,C 180,E1 4532.72,E2 4532.72} C_VEL
LIN {X 0,Y 522.258,Z 580.66,A -85,B 0,C 180,E1 4538.487,E2 4538.487} C_VEL
LIN {X 0,Y 522.381,Z 580.66,A -85,B 0,C 180,E1 4544.068,E2 4544.068} C_VEL
LIN {X 0,Y 522.406,Z 580.66,A -85,B 0,C 180,E1 4550.385,E2 4550.385} C_VEL
LIN {X 0,Y 522.369,Z 580.66,A -85,B 0,C 180,E1 4556.584,E2 4556.584} C_VEL
LIN {X 0,Y 522.545,Z 580.66,A -85,B 0,C 180,E1 4559.754,E2 4559.754} C_VEL
LIN {X 0,Y 533.314,Z 608.839,A -85,B 0,C 180,E1 4560.729,E2 4560.729} C_VEL
LIN {X 0,Y 532.429,Z 668.906,A -85,B 0,C 180,E1 4561.751,E2 4561.751} C_VEL
LIN {X 0,Y 531.127,Z 704.669,A -85,B 0,C 180,E1 4563.008,E2 4563.008} C_VEL
LIN {X 0,Y 529.348,Z 739.96,A -85,B 0,C 180,E1 4564.932,E2 4564.932} C_VEL
LIN {X 0,Y 527.465,Z 772.845,A -85,B 0,C 180,E1 4567.491,E2 4567.491} C_VEL
LIN {X 0,Y 525.837,Z 800.736,A -85,B 0,C 180,E1 4570.443,E2 4570.443} C_VEL
LIN {X 0,Y 524.522,Z 824.958,A -85,B 0,C 180,E1 4573.868,E2 4573.868} C_VEL
LIN {X 0,Y 523.769,Z 843.714,A -85,B 0,C 180,E1 4577.477,E2 4577.477} C_VEL
LIN {X 0,Y 523.39,Z 857.455,A -85,B 0,C 180,E1 4581.263,E2 4581.263} C_VEL
LIN {X 0,Y 523.201,Z 865.962,A -85,B 0,C 180,E1 4585.018,E2 4585.018} C_VEL
LIN {X 0,Y 523.134,Z 869.509,A -85,B 0,C 180,E1 4588.34,E2 4588.34} C_VEL
LIN {X 0,Y 523.204,Z 869.511,A -85,B 0,C 180,E1 4591.657,E2 4591.657} C_VEL
LIN {X 0,Y 523.261,Z 865.968,A -85,B 0,C 180,E1 4594.978,E2 4594.978} C_VEL
LIN {X 0,Y 523.397,Z 856.178,A -85,B 0,C 180,E1 4599.153,E2 4599.153} C_VEL
LIN {X 0,Y 523.81,Z 841.782,A -85,B 0,C 180,E1 4602.943,E2 4602.943} C_VEL
LIN {X 0,Y 524.603,Z 822.325,A -85,B 0,C 180,E1 4606.557,E2 4606.557} C_VEL
LIN {X 0,Y 526.006,Z 797.249,A -85,B 0,C 180,E1 4609.985,E2 4609.985} C_VEL
LIN {X 0,Y 527.773,Z 767.481,A -85,B 0,C 180,E1 4612.983,E2 4612.983} C_VEL
LIN {X 0,Y 529.679,Z 734.902,A -85,B 0,C 180,E1 4615.387,E2 4615.387} C_VEL
LIN {X 0,Y 531.412,Z 700.226,A -85,B 0,C 180,E1 4617.186,E2 4617.186} C_VEL
LIN {X 0,Y 532.652,Z 664.565,A -85,B 0,C 180,E1 4618.354,E2 4618.354} C_VEL
LIN {X 0,Y 532.651,Z 605.13,A -85,B 0,C 180,E1 4619.362,E2 4619.362} C_VEL
LIN {X 0,Y 522.53,Z 580.66,A -85,B 0,C 180,E1 4620.296,E2 4620.296} C_VEL
LIN {X 0,Y 522.303,Z 580.66,A -85,B 0,C 180,E1 4625.75,E2 4625.75} C_VEL
LIN {X 0,Y 522.304,Z 580.66,A -85,B 0,C 180,E1 4631.811,E2 4631.811} C_VEL
LIN {X 0,Y 522.424,Z 580.66,A -85,B 0,C 180,E1 4638.204,E2 4638.204} C_VEL
LIN {X 0,Y 522.322,Z 580.66,A -85,B 0,C 180,E1 4644.574,E2 4644.574} C_VEL
LIN {X 0,Y 522.389,Z 580.66,A -85,B 0,C 180,E1 4650.487,E2 4650.487} C_VEL
LIN {X 0,Y 522.543,Z 580.66,A -85,B 0,C 180,E1 4656.074,E2 4656.074} C_VEL
LIN {X 0,Y 522.709,Z 580.66,A -85,B 0,C 180,E1 4661.426,E2 4661.426} C_VEL
LIN {X 0,Y 522.619,Z 580.66,A -85,B 0,C 180,E1 4668.305,E2 4668.305} C_VEL
LIN {X 0,Y 522.904,Z 580.66,A -85,B 0,C 180,E1 4673.354,E2 4673.354} C_VEL
LIN {X 0,Y 522.902,Z 580.66,A -85,B 0,C 180,E1 4680.005,E2 4680.005} C_VEL
LIN {X 0,Y 522.847,Z 580.66,A -85,B 0,C 180,E1 4684.988,E2 4684.988} C_VEL
LIN {X 0,Y 522.744,Z 580.66,A -85,B 0,C 180,E1 4690.031,E2 4690.031} C_VEL
LIN {X 0,Y 522.669,Z 580.66,A -85,B 0,C 180,E1 4695.117,E2 4695.117} C_VEL
LIN {X 0,Y 522.606,Z 580.66,A -85,B 0,C 180,E1 4700.348,E2 4700.348} C_VEL
LIN {X 0,Y 522.436,Z 580.66,A -85,B 0,C 180,E1 4706.058,E2 4706.058} C_VEL
LIN {X 0,Y 522.42,Z 580.66,A -85,B 0,C 180,E1 4711.449,E2 4711.449} C_VEL
LIN {X 0,Y 522.392,Z 580.66,A -85,B 0,C 180,E1 4717.497,E2 4717.497} C_VEL
LIN {X 0,Y 522.231,Z 580.66,A -85,B 0,C 180,E1 4723.551,E2 4723.551} C_VEL
LIN {X 0,Y 522.37,Z 580.66,A -85,B 0,C 180,E1 4728.908,E2 4728.908} C_VEL
LIN {X 0,Y 522.488,Z 580.66,A -85,B 0,C 180,E1 4734.584,E2 4734.584} C_VEL
LIN {X 0,Y 522.444,Z 580.66,A -85,B 0,C 180,E1 4740.487,E2 4740.487} C_VEL
LIN {X 0,Y 522.621,Z 580.925,A -85,B 0,C 180,E1 4746.827,E2 4746.827} C_VEL
LIN {X 0,Y 529.391,Z 604.365,A -85,B 0,C 180,E1 4748.459,E2 4748.459} C_VEL
LIN {X 0,Y 527.812,Z 634.013,A -85,B 0,C 180,E1 4750.523,E2 4750.523} C_VEL
LIN {X 0,Y 526.131,Z 659.588,A -85,B 0,C 180,E1 4753.062,E2 4753.062} C_VEL
LIN {X 0,Y 524.745,Z 681.641,A -85,B 0,C 180,E1 4756.098,E2 4756.098} C_VEL
LIN {X 0,Y 523.792,Z 699.727,A -85,B 0,C 180,E1 4759.651,E2 4759.651} C_VEL
LIN {X 0,Y 523.392,Z 711.903,A -85,B 0,C 180,E1 4763.357,E2 4763.357} C_VEL
LIN {X 0,Y 523.255,Z 718.085,A -85,B 0,C 180,E1 4766.684,E2 4766.684} C_VEL
LIN {X 0,Y 523.216,Z 720.069,A -85,B 0,C 180,E1 4770.002,E2 4770.002} C_VEL
LIN {X 0,Y 523.276,Z 717.104,A -85,B 0,C 180,E1 4773.942,E2 4773.942} C_VEL
LIN {X 0,Y 523.512,Z 708.154,A -85,B 0,C 180,E1 4777.897,E2 4777.897} C_VEL
LIN {X 0,Y 524.057,Z 694.883,A -85,B 0,C 180,E1 4781.349,E2 4781.349} C_VEL
LIN {X 0,Y 525.157,Z 675.109,A -85,B 0,C 180,E1 4784.825,E2 4784.825} C_VEL
LIN {X 0,Y 526.688,Z 651.116,A -85,B 0,C 180,E1 4787.785,E2 4787.785} C_VEL
LIN {X 0,Y 528.364,Z 624.75,A -85,B 0,C 180,E1 4790.114,E2 4790.114} C_VEL
LIN {X 0,Y 528.826,Z 600.254,A -85,B 0,C 180,E1 4791.727,E2 4791.727} C_VEL
LIN {X 0,Y 522.621,Z 580.66,A -85,B 0,C 180,E1 4793.17,E2 4793.17} C_VEL
LIN {X 0,Y 522.386,Z 580.66,A -85,B 0,C 180,E1 4799.591,E2 4799.591} C_VEL
LIN {X 0,Y 522.362,Z 580.66,A -85,B 0,C 180,E1 4805.744,E2 4805.744} C_VEL
LIN {X 0,Y 522.334,Z 580.66,A -85,B 0,C 180,E1 4811.813,E2 4811.813} C_VEL
LIN {X 0,Y 522.37,Z 580.66,A -85,B 0,C 180,E1 4818.186,E2 4818.186} C_VEL
LIN {X 0,Y 522.287,Z 580.66,A -85,B 0,C 180,E1 4824.56,E2 4824.56} C_VEL
LIN {X 0,Y 522.365,Z 580.66,A -85,B 0,C 180,E1 4830.475,E2 4830.475} C_VEL
LIN {X 0,Y 522.562,Z 580.66,A -85,B 0,C 180,E1 4836.065,E2 4836.065} C_VEL
LIN {X 0,Y 522.718,Z 580.66,A -85,B 0,C 180,E1 4841.416,E2 4841.416} C_VEL
LIN {X 0,Y 522.584,Z 580.66,A -85,B 0,C 180,E1 4848.294,E2 4848.294} C_VEL
LIN {X 0,Y 522.933,Z 580.66,A -85,B 0,C 180,E1 4853.345,E2 4853.345} C_VEL
LIN {X 0,Y 522.928,Z 580.66,A -85,B 0,C 180,E1 4859.995,E2 4859.995} C_VEL
LIN {X 0,Y 522.85,Z 580.66,A -85,B 0,C 180,E1 4864.979,E2 4864.979} C_VEL
LIN {X 0,Y 522.757,Z 580.66,A -85,B 0,C 180,E1 4870.022,E2 4870.022} C_VEL
LIN {X 0,Y 522.675,Z 580.66,A -85,B 0,C 180,E1 4875.107,E2 4875.107} C_VEL
LIN {X 0,Y 522.604,Z 580.66,A -85,B 0,C 180,E1 4880.339,E2 4880.339} C_VEL
LIN {X 0,Y 522.45,Z 580.66,A -85,B 0,C 180,E1 4886.054,E2 4886.054} C_VEL
LIN {X 0,Y 522.356,Z 580.66,A -85,B 0,C 180,E1 4891.442,E2 4891.442} C_VEL
LIN {X 0,Y 522.386,Z 580.66,A -85,B 0,C 180,E1 4892.72,E2 4892.72} C_VEL
